Yaskawa INFORM job: DEMO_ROOF_UPPER_0625_3PAINT_27.JBI

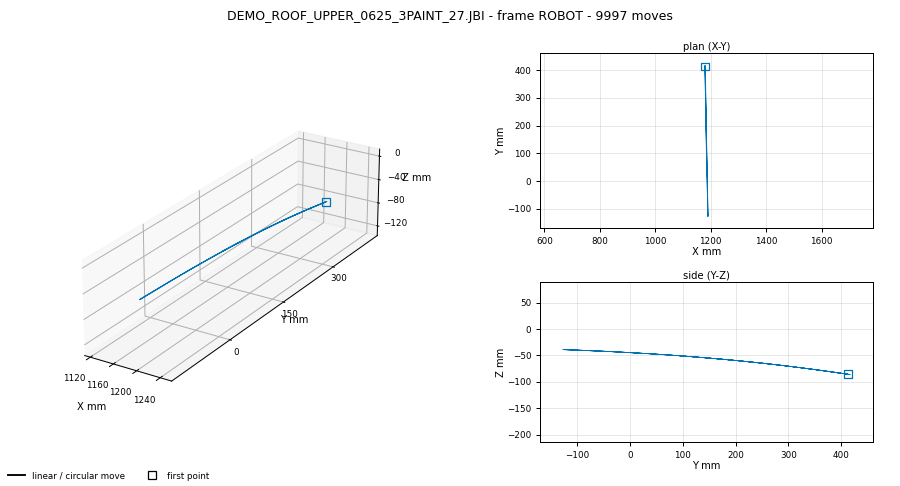
[picture p0: tool path of DEMO_ROOF_UPPER_0625_3PAINT_27.JBI in frame ROBOT, 9997 of 9997 moves have a stored position in this frame; points joined in program order, loops and branches not executed]
/JOB
//NAME DEMO_ROOF_UPPER_0625_3PAINT27
//POS
///NPOS 9997,0,0,0,0,0
///TOOL 0
///USER 0
///POSTYPE ROBOT
///RECTAN
///RCONF 1,0,0,0,0,0,0,0,0,0,0,0,0,0,0,0,0,0,0,0,0,0,0,0
C00000=1180.489,413.583,-85.570,-176.011,9.119,148.688
C00001=1180.493,413.335,-85.534,-176.011,9.117,148.687
C00002=1180.497,413.087,-85.498,-176.011,9.115,148.686
C00003=1180.501,412.840,-85.462,-176.011,9.113,148.686
C00004=1180.505,412.594,-85.426,-176.010,9.111,148.686
C00005=1180.509,412.346,-85.390,-176.010,9.109,148.685
C00006=1180.513,412.098,-85.354,-176.010,9.107,148.684
C00007=1180.517,411.851,-85.319,-176.010,9.105,148.684
C00008=1180.521,411.603,-85.282,-176.011,9.103,148.683
C00009=1180.525,411.356,-85.246,-176.010,9.101,148.683
C00010=1180.528,411.108,-85.211,-176.010,9.099,148.682
C00011=1180.532,410.861,-85.174,-176.010,9.097,148.682
C00012=1180.536,410.614,-85.138,-176.010,9.095,148.681
C00013=1180.540,410.367,-85.103,-176.009,9.093,148.680
C00014=1180.545,410.119,-85.067,-176.010,9.091,148.680
C00015=1180.548,409.872,-85.031,-176.009,9.089,148.679
C00016=1180.553,409.625,-84.995,-176.009,9.087,148.679
C00017=1180.556,409.377,-84.959,-176.009,9.085,148.678
C00018=1180.560,409.130,-84.924,-176.009,9.082,148.678
C00019=1180.564,408.882,-84.887,-176.009,9.081,148.677
C00020=1180.568,408.635,-84.851,-176.009,9.079,148.677
C00021=1180.572,408.388,-84.816,-176.009,9.076,148.676
C00022=1180.576,408.140,-84.780,-176.009,9.075,148.675
C00023=1180.580,407.893,-84.744,-176.009,9.072,148.675
C00024=1180.583,407.646,-84.708,-176.009,9.070,148.674
C00025=1180.588,407.398,-84.672,-176.009,9.068,148.674
C00026=1180.591,407.151,-84.636,-176.008,9.066,148.673
C00027=1180.595,406.903,-84.601,-176.009,9.064,148.672
C00028=1180.599,406.655,-84.565,-176.008,9.062,148.672
C00029=1180.603,406.409,-84.529,-176.008,9.060,148.671
C00030=1180.607,406.162,-84.493,-176.008,9.057,148.671
C00031=1180.611,405.914,-84.457,-176.008,9.056,148.670
C00032=1180.615,405.666,-84.422,-176.008,9.053,148.670
C00033=1180.619,405.419,-84.386,-176.008,9.051,148.669
C00034=1180.623,405.171,-84.350,-176.008,9.048,148.668
C00035=1180.627,404.924,-84.314,-176.008,9.047,148.668
C00036=1180.631,404.677,-84.278,-176.008,9.044,148.667
C00037=1180.635,404.429,-84.242,-176.008,9.042,148.667
C00038=1180.639,404.182,-84.207,-176.008,9.040,148.666
C00039=1180.643,403.934,-84.171,-176.008,9.037,148.665
C00040=1180.647,403.687,-84.135,-176.007,9.036,148.665
C00041=1180.650,403.440,-84.099,-176.008,9.033,148.664
C00042=1180.655,403.193,-84.064,-176.007,9.031,148.664
C00043=1180.659,402.945,-84.027,-176.008,9.029,148.663
C00044=1180.663,402.698,-83.992,-176.007,9.026,148.662
C00045=1180.666,402.450,-83.956,-176.008,9.024,148.662
C00046=1180.670,402.203,-83.921,-176.008,9.021,148.661
C00047=1180.674,401.955,-83.885,-176.007,9.020,148.661
C00048=1180.678,401.709,-83.849,-176.007,9.017,148.660
C00049=1180.682,401.461,-83.813,-176.007,9.015,148.659
C00050=1180.686,401.213,-83.777,-176.007,9.012,148.659
C00051=1180.690,400.966,-83.741,-176.007,9.010,148.658
C00052=1180.694,400.718,-83.706,-176.007,9.007,148.657
C00053=1180.697,400.471,-83.670,-176.008,9.005,148.657
C00054=1180.702,400.224,-83.635,-176.007,9.003,148.656
C00055=1180.706,399.976,-83.599,-176.008,9.000,148.656
C00056=1180.710,399.729,-83.564,-176.007,8.998,148.655
C00057=1180.714,399.481,-83.527,-176.008,8.996,148.654
C00058=1180.718,399.233,-83.492,-176.008,8.993,148.654
C00059=1180.721,398.987,-83.456,-176.007,8.990,148.653
C00060=1180.725,398.740,-83.420,-176.008,8.988,148.652
C00061=1180.730,398.492,-83.384,-176.007,8.986,148.652
C00062=1180.733,398.244,-83.349,-176.008,8.983,148.651
C00063=1180.737,397.997,-83.313,-176.008,8.981,148.650
C00064=1180.741,397.749,-83.278,-176.008,8.978,148.650
C00065=1180.746,397.502,-83.242,-176.008,8.976,148.649
C00066=1180.749,397.255,-83.206,-176.008,8.974,148.649
C00067=1180.753,397.007,-83.171,-176.008,8.970,148.648
C00068=1180.757,396.760,-83.135,-176.008,8.968,148.647
C00069=1180.761,396.512,-83.099,-176.008,8.965,148.647
C00070=1180.765,396.265,-83.064,-176.008,8.963,148.646
C00071=1180.769,396.018,-83.028,-176.008,8.961,148.645
C00072=1180.773,395.770,-82.993,-176.008,8.958,148.645
C00073=1180.776,395.523,-82.957,-176.009,8.955,148.644
C00074=1180.781,395.276,-82.921,-176.009,8.952,148.643
C00075=1180.785,395.028,-82.886,-176.009,8.950,148.643
C00076=1180.789,394.781,-82.850,-176.009,8.948,148.642
C00077=1180.792,394.533,-82.815,-176.009,8.945,148.641
C00078=1180.797,394.285,-82.779,-176.010,8.942,148.641
C00079=1180.801,394.038,-82.743,-176.009,8.939,148.640
C00080=1180.805,393.791,-82.708,-176.010,8.937,148.640
C00081=1180.808,393.543,-82.672,-176.010,8.934,148.639
C00082=1180.812,393.296,-82.637,-176.010,8.931,148.638
C00083=1180.816,393.048,-82.601,-176.010,8.929,148.638
C00084=1180.821,392.801,-82.565,-176.011,8.926,148.637
C00085=1180.824,392.554,-82.530,-176.011,8.923,148.636
C00086=1180.829,392.269,-82.490,-176.011,8.920,148.636
C00087=1180.833,391.986,-82.449,-176.012,8.916,148.635
C00088=1180.838,391.701,-82.408,-176.011,8.914,148.634
C00089=1180.842,391.417,-82.367,-176.012,8.911,148.633
C00090=1180.846,391.169,-82.332,-176.013,8.907,148.633
C00091=1180.850,390.922,-82.297,-176.013,8.905,148.632
C00092=1180.854,390.675,-82.261,-176.013,8.902,148.631
C00093=1180.859,390.427,-82.225,-176.014,8.899,148.631
C00094=1180.862,390.180,-82.190,-176.014,8.896,148.630
C00095=1180.866,389.933,-82.154,-176.014,8.894,148.630
C00096=1180.870,389.685,-82.119,-176.015,8.890,148.629
C00097=1180.874,389.438,-82.083,-176.015,8.888,148.628
C00098=1180.878,389.190,-82.049,-176.015,8.885,148.627
C00099=1180.882,388.943,-82.013,-176.016,8.882,148.627
C00100=1180.886,388.695,-81.978,-176.016,8.879,148.626
C00101=1180.890,388.448,-81.942,-176.017,8.876,148.626
C00102=1180.894,388.200,-81.906,-176.018,8.873,148.625
C00103=1180.898,387.953,-81.871,-176.017,8.870,148.624
C00104=1180.902,387.705,-81.836,-176.018,8.867,148.624
C00105=1180.906,387.458,-81.801,-176.019,8.864,148.623
C00106=1180.910,387.211,-81.765,-176.019,8.861,148.622
C00107=1180.914,386.963,-81.730,-176.020,8.858,148.622
C00108=1180.917,386.716,-81.694,-176.020,8.855,148.621
C00109=1180.921,386.468,-81.659,-176.021,8.852,148.620
C00110=1180.925,386.221,-81.624,-176.022,8.849,148.620
C00111=1180.929,385.973,-81.589,-176.022,8.845,148.619
C00112=1180.933,385.726,-81.553,-176.022,8.843,148.619
C00113=1180.938,385.478,-81.518,-176.023,8.840,148.618
C00114=1180.942,385.231,-81.483,-176.024,8.837,148.617
C00115=1180.945,384.983,-81.447,-176.024,8.834,148.617
C00116=1180.949,384.736,-81.411,-176.025,8.830,148.616
C00117=1180.954,384.488,-81.377,-176.026,8.827,148.615
C00118=1180.957,384.241,-81.341,-176.027,8.824,148.615
C00119=1180.961,383.993,-81.306,-176.028,8.821,148.614
C00120=1180.966,383.746,-81.271,-176.028,8.818,148.614
C00121=1180.969,383.498,-81.236,-176.029,8.815,148.613
C00122=1180.973,383.251,-81.200,-176.030,8.812,148.612
C00123=1180.977,383.003,-81.166,-176.031,8.809,148.612
C00124=1180.981,382.756,-81.130,-176.031,8.805,148.611
C00125=1180.985,382.508,-81.095,-176.032,8.802,148.611
C00126=1180.989,382.261,-81.060,-176.033,8.799,148.610
C00127=1180.993,382.014,-81.025,-176.034,8.795,148.609
C00128=1180.997,381.766,-80.989,-176.035,8.792,148.609
C00129=1181.001,381.519,-80.955,-176.036,8.789,148.608
C00130=1181.005,381.271,-80.919,-176.036,8.786,148.607
C00131=1181.009,381.024,-80.885,-176.037,8.783,148.607
C00132=1181.013,380.776,-80.849,-176.038,8.780,148.606
C00133=1181.017,380.529,-80.814,-176.039,8.776,148.606
C00134=1181.021,380.281,-80.779,-176.040,8.773,148.605
C00135=1181.025,380.034,-80.744,-176.041,8.769,148.604
C00136=1181.029,379.786,-80.709,-176.042,8.766,148.604
C00137=1181.033,379.539,-80.674,-176.044,8.763,148.603
C00138=1181.036,379.291,-80.639,-176.045,8.760,148.603
C00139=1181.040,379.044,-80.604,-176.045,8.757,148.602
C00140=1181.045,378.796,-80.569,-176.047,8.753,148.602
C00141=1181.048,378.549,-80.534,-176.048,8.750,148.601
C00142=1181.053,378.301,-80.499,-176.048,8.746,148.601
C00143=1181.057,378.054,-80.464,-176.050,8.743,148.600
C00144=1181.061,377.806,-80.429,-176.051,8.740,148.599
C00145=1181.065,377.559,-80.394,-176.052,8.736,148.599
C00146=1181.069,377.311,-80.359,-176.053,8.733,148.598
C00147=1181.073,377.064,-80.324,-176.054,8.730,148.598
C00148=1181.076,376.816,-80.290,-176.055,8.726,148.597
C00149=1181.081,376.569,-80.254,-176.057,8.723,148.597
C00150=1181.085,376.321,-80.220,-176.058,8.719,148.596
C00151=1181.088,376.073,-80.185,-176.059,8.716,148.595
C00152=1181.093,375.826,-80.150,-176.061,8.712,148.595
C00153=1181.097,375.578,-80.115,-176.062,8.709,148.594
C00154=1181.101,375.331,-80.080,-176.063,8.705,148.594
C00155=1181.104,375.083,-80.045,-176.064,8.702,148.593
C00156=1181.109,374.836,-80.011,-176.066,8.699,148.593
C00157=1181.112,374.589,-79.975,-176.066,8.695,148.592
C00158=1181.116,374.340,-79.940,-176.068,8.692,148.592
C00159=1181.121,374.093,-79.906,-176.070,8.688,148.591
C00160=1181.124,373.846,-79.871,-176.071,8.685,148.591
C00161=1181.128,373.598,-79.837,-176.072,8.681,148.590
C00162=1181.132,373.350,-79.802,-176.073,8.678,148.590
C00163=1181.137,373.103,-79.767,-176.075,8.674,148.589
C00164=1181.140,372.856,-79.732,-176.077,8.671,148.589
C00165=1181.145,372.608,-79.698,-176.077,8.668,148.588
C00166=1181.148,372.360,-79.663,-176.079,8.664,148.588
C00167=1181.153,372.113,-79.629,-176.081,8.661,148.587
C00168=1181.156,371.866,-79.594,-176.082,8.657,148.587
C00169=1181.161,371.618,-79.559,-176.084,8.654,148.586
C00170=1181.165,371.370,-79.524,-176.085,8.650,148.586
C00171=1181.169,371.123,-79.490,-176.087,8.646,148.585
C00172=1181.172,370.875,-79.455,-176.088,8.643,148.585
C00173=1181.177,370.628,-79.420,-176.090,8.640,148.584
C00174=1181.181,370.380,-79.386,-176.091,8.636,148.584
C00175=1181.184,370.133,-79.352,-176.093,8.633,148.583
C00176=1181.188,369.885,-79.317,-176.095,8.630,148.583
C00177=1181.193,369.637,-79.282,-176.096,8.626,148.582
C00178=1181.196,369.389,-79.248,-176.098,8.622,148.582
C00179=1181.200,369.143,-79.213,-176.100,8.618,148.581
C00180=1181.204,368.894,-79.178,-176.101,8.616,148.581
C00181=1181.208,368.647,-79.144,-176.103,8.612,148.581
C00182=1181.212,368.399,-79.109,-176.104,8.608,148.580
C00183=1181.217,368.152,-79.075,-176.106,8.604,148.580
C00184=1181.221,367.905,-79.041,-176.108,8.601,148.579
C00185=1181.225,367.657,-79.006,-176.109,8.598,148.579
C00186=1181.229,367.409,-78.972,-176.111,8.594,148.578
C00187=1181.232,367.161,-78.938,-176.113,8.591,148.578
C00188=1181.237,366.914,-78.903,-176.114,8.587,148.577
C00189=1181.240,366.666,-78.869,-176.116,8.584,148.577
C00190=1181.245,366.384,-78.829,-176.118,8.580,148.577
C00191=1181.249,366.103,-78.791,-176.120,8.575,148.576
C00192=1181.254,365.821,-78.752,-176.122,8.572,148.576
C00193=1181.258,365.540,-78.713,-176.125,8.567,148.575
C00194=1181.263,365.292,-78.678,-176.126,8.564,148.575
C00195=1181.267,365.045,-78.645,-176.128,8.561,148.574
C00196=1181.271,364.797,-78.610,-176.129,8.557,148.574
C00197=1181.275,364.550,-78.575,-176.131,8.554,148.573
C00198=1181.279,364.302,-78.541,-176.133,8.550,148.573
C00199=1181.283,364.054,-78.507,-176.135,8.547,148.573
C00200=1181.287,363.807,-78.473,-176.137,8.543,148.572
C00201=1181.291,363.558,-78.439,-176.139,8.540,148.572
C00202=1181.295,363.311,-78.405,-176.141,8.536,148.572
C00203=1181.298,363.064,-78.371,-176.143,8.532,148.571
C00204=1181.303,362.816,-78.336,-176.144,8.529,148.571
C00205=1181.307,362.569,-78.302,-176.147,8.525,148.570
C00206=1181.311,362.320,-78.268,-176.149,8.522,148.570
C00207=1181.315,362.073,-78.234,-176.150,8.518,148.570
C00208=1181.319,361.826,-78.200,-176.153,8.515,148.569
C00209=1181.323,361.578,-78.165,-176.154,8.511,148.569
C00210=1181.328,361.330,-78.132,-176.156,8.508,148.568
C00211=1181.331,361.083,-78.098,-176.159,8.504,148.568
C00212=1181.335,360.835,-78.064,-176.160,8.501,148.568
C00213=1181.339,360.588,-78.029,-176.162,8.497,148.567
C00214=1181.343,360.340,-77.996,-176.164,8.494,148.567
C00215=1181.347,360.092,-77.961,-176.166,8.490,148.567
C00216=1181.351,359.845,-77.927,-176.169,8.487,148.567
C00217=1181.355,359.597,-77.894,-176.170,8.483,148.566
C00218=1181.360,359.349,-77.860,-176.173,8.480,148.566
C00219=1181.363,359.101,-77.826,-176.174,8.476,148.565
C00220=1181.367,358.854,-77.792,-176.177,8.473,148.565
C00221=1181.372,358.606,-77.758,-176.178,8.469,148.565
C00222=1181.375,358.358,-77.724,-176.181,8.466,148.565
C00223=1181.379,358.111,-77.690,-176.183,8.462,148.564
C00224=1181.384,357.863,-77.657,-176.185,8.459,148.564
C00225=1181.388,357.616,-77.623,-176.187,8.456,148.564
C00226=1181.391,357.367,-77.589,-176.189,8.451,148.563
C00227=1181.396,357.120,-77.555,-176.192,8.448,148.563
C00228=1181.400,356.872,-77.522,-176.194,8.444,148.563
C00229=1181.404,356.625,-77.488,-176.196,8.441,148.562
C00230=1181.407,356.377,-77.454,-176.198,8.438,148.562
C00231=1181.412,356.129,-77.420,-176.200,8.434,148.562
C00232=1181.416,355.882,-77.387,-176.202,8.431,148.561
C00233=1181.420,355.634,-77.353,-176.204,8.428,148.561
C00234=1181.424,355.387,-77.320,-176.206,8.424,148.561
C00235=1181.428,355.139,-77.285,-176.208,8.421,148.561
C00236=1181.432,354.891,-77.252,-176.211,8.417,148.560
C00237=1181.436,354.643,-77.218,-176.213,8.414,148.560
C00238=1181.440,354.396,-77.185,-176.215,8.410,148.560
C00239=1181.444,354.148,-77.151,-176.217,8.407,148.559
C00240=1181.449,353.899,-77.117,-176.219,8.404,148.559
C00241=1181.452,353.652,-77.083,-176.221,8.400,148.559
C00242=1181.457,353.405,-77.050,-176.224,8.396,148.559
C00243=1181.461,353.157,-77.017,-176.226,8.393,148.558
C00244=1181.465,352.910,-76.983,-176.229,8.389,148.558
C00245=1181.469,352.662,-76.950,-176.230,8.386,148.558
C00246=1181.473,352.413,-76.916,-176.233,8.382,148.557
C00247=1181.477,352.166,-76.883,-176.235,8.379,148.557
C00248=1181.481,351.919,-76.849,-176.237,8.376,148.557
C00249=1181.485,351.671,-76.816,-176.239,8.372,148.557
C00250=1181.489,351.423,-76.783,-176.241,8.369,148.556
C00251=1181.493,351.175,-76.750,-176.243,8.366,148.556
C00252=1181.497,350.928,-76.716,-176.246,8.362,148.556
C00253=1181.501,350.680,-76.682,-176.248,8.359,148.556
C00254=1181.505,350.432,-76.649,-176.250,8.356,148.556
C00255=1181.510,350.184,-76.615,-176.253,8.352,148.555
C00256=1181.514,349.936,-76.582,-176.254,8.349,148.555
C00257=1181.518,349.689,-76.549,-176.257,8.345,148.555
C00258=1181.522,349.441,-76.516,-176.259,8.342,148.554
C00259=1181.526,349.193,-76.483,-176.261,8.339,148.554
C00260=1181.530,348.946,-76.449,-176.263,8.335,148.554
C00261=1181.534,348.698,-76.416,-176.266,8.332,148.554
C00262=1181.538,348.451,-76.382,-176.268,8.329,148.554
C00263=1181.543,348.203,-76.349,-176.270,8.325,148.553
C00264=1181.547,347.955,-76.316,-176.273,8.321,148.553
C00265=1181.550,347.707,-76.283,-176.275,8.318,148.553
C00266=1181.554,347.459,-76.249,-176.278,8.315,148.553
C00267=1181.559,347.211,-76.216,-176.279,8.311,148.552
C00268=1181.563,346.963,-76.183,-176.282,8.308,148.552
C00269=1181.567,346.716,-76.150,-176.284,8.304,148.552
C00270=1181.571,346.468,-76.117,-176.286,8.301,148.552
C00271=1181.575,346.220,-76.084,-176.288,8.298,148.551
C00272=1181.579,345.973,-76.050,-176.291,8.294,148.551
C00273=1181.584,345.724,-76.018,-176.293,8.291,148.551
C00274=1181.587,345.477,-75.985,-176.295,8.288,148.551
C00275=1181.591,345.229,-75.952,-176.297,8.285,148.550
C00276=1181.595,344.981,-75.919,-176.300,8.281,148.550
C00277=1181.599,344.734,-75.886,-176.302,8.278,148.550
C00278=1181.604,344.486,-75.853,-176.304,8.275,148.550
C00279=1181.608,344.238,-75.820,-176.307,8.272,148.550
C00280=1181.612,343.990,-75.787,-176.309,8.268,148.550
C00281=1181.616,343.742,-75.754,-176.311,8.265,148.549
C00282=1181.620,343.494,-75.721,-176.314,8.262,148.549
C00283=1181.624,343.247,-75.688,-176.316,8.258,148.549
C00284=1181.628,342.999,-75.655,-176.318,8.255,148.549
C00285=1181.632,342.751,-75.623,-176.320,8.252,148.549
C00286=1181.637,342.503,-75.590,-176.323,8.248,148.548
C00287=1181.641,342.256,-75.557,-176.325,8.245,148.548
C00288=1181.645,342.008,-75.524,-176.327,8.242,148.548
C00289=1181.649,341.760,-75.492,-176.330,8.238,148.548
C00290=1181.653,341.513,-75.459,-176.332,8.235,148.547
C00291=1181.657,341.265,-75.426,-176.335,8.232,148.547
C00292=1181.662,341.016,-75.393,-176.337,8.229,148.547
C00293=1181.666,340.769,-75.360,-176.339,8.226,148.547
C00294=1181.670,340.490,-75.323,-176.342,8.221,148.547
C00295=1181.674,340.211,-75.286,-176.344,8.218,148.547
C00296=1181.680,339.931,-75.250,-176.347,8.214,148.546
C00297=1181.684,339.653,-75.213,-176.350,8.211,148.546
C00298=1181.688,339.405,-75.180,-176.352,8.208,148.546
C00299=1181.693,339.157,-75.148,-176.354,8.204,148.546
C00300=1181.696,338.909,-75.115,-176.356,8.201,148.546
C00301=1181.700,338.662,-75.082,-176.359,8.198,148.545
C00302=1181.705,338.413,-75.050,-176.361,8.194,148.545
C00303=1181.709,338.167,-75.017,-176.364,8.191,148.545
C00304=1181.713,337.918,-74.985,-176.366,8.188,148.545
C00305=1181.717,337.671,-74.952,-176.368,8.185,148.545
C00306=1181.721,337.422,-74.920,-176.370,8.181,148.545
C00307=1181.726,337.174,-74.888,-176.373,8.178,148.545
C00308=1181.730,336.926,-74.854,-176.375,8.175,148.544
C00309=1181.733,336.678,-74.823,-176.378,8.172,148.544
C00310=1181.738,336.431,-74.790,-176.380,8.168,148.544
C00311=1181.742,336.183,-74.758,-176.383,8.165,148.544
C00312=1181.746,335.936,-74.725,-176.385,8.162,148.544
C00313=1181.750,335.687,-74.692,-176.387,8.159,148.543
C00314=1181.754,335.439,-74.661,-176.389,8.156,148.543
C00315=1181.758,335.191,-74.627,-176.392,8.153,148.543
C00316=1181.763,334.944,-74.596,-176.394,8.149,148.543
C00317=1181.767,334.696,-74.563,-176.397,8.146,148.543
C00318=1181.770,334.448,-74.531,-176.399,8.143,148.543
C00319=1181.775,334.200,-74.498,-176.402,8.140,148.543
C00320=1181.779,333.953,-74.467,-176.404,8.136,148.542
C00321=1181.783,333.705,-74.434,-176.406,8.133,148.542
C00322=1181.788,333.457,-74.401,-176.409,8.130,148.542
C00323=1181.792,333.209,-74.370,-176.411,8.127,148.542
C00324=1181.796,332.960,-74.337,-176.413,8.123,148.542
C00325=1181.800,332.713,-74.305,-176.416,8.120,148.542
C00326=1181.804,332.465,-74.273,-176.418,8.117,148.542
C00327=1181.808,332.217,-74.241,-176.421,8.114,148.541
C00328=1181.812,331.969,-74.209,-176.423,8.111,148.541
C00329=1181.817,331.721,-74.177,-176.426,8.107,148.541
C00330=1181.820,331.474,-74.144,-176.428,8.104,148.541
C00331=1181.825,331.226,-74.112,-176.431,8.101,148.541
C00332=1181.828,330.978,-74.080,-176.433,8.098,148.541
C00333=1181.833,330.730,-74.048,-176.435,8.094,148.541
C00334=1181.837,330.482,-74.016,-176.438,8.091,148.541
C00335=1181.841,330.234,-73.984,-176.440,8.088,148.540
C00336=1181.846,329.986,-73.952,-176.443,8.085,148.540
C00337=1181.850,329.738,-73.920,-176.445,8.083,148.540
C00338=1181.854,329.490,-73.888,-176.447,8.079,148.540
C00339=1181.858,329.242,-73.856,-176.449,8.076,148.540
C00340=1181.862,328.994,-73.824,-176.452,8.073,148.540
C00341=1181.867,328.746,-73.792,-176.454,8.070,148.540
C00342=1181.870,328.498,-73.760,-176.457,8.067,148.540
C00343=1181.875,328.251,-73.729,-176.459,8.063,148.539
C00344=1181.879,328.002,-73.696,-176.462,8.060,148.539
C00345=1181.883,327.754,-73.664,-176.464,8.057,148.539
C00346=1181.887,327.507,-73.633,-176.467,8.054,148.539
C00347=1181.891,327.259,-73.600,-176.469,8.051,148.539
C00348=1181.896,327.011,-73.569,-176.472,8.048,148.539
C00349=1181.899,326.763,-73.537,-176.474,8.044,148.539
C00350=1181.904,326.515,-73.505,-176.476,8.041,148.539
C00351=1181.908,326.268,-73.473,-176.479,8.038,148.539
C00352=1181.912,326.020,-73.441,-176.481,8.035,148.538
C00353=1181.916,325.772,-73.409,-176.484,8.032,148.538
C00354=1181.921,325.523,-73.378,-176.486,8.028,148.538
C00355=1181.925,325.275,-73.346,-176.489,8.025,148.538
C00356=1181.929,325.028,-73.315,-176.491,8.022,148.538
C00357=1181.933,324.780,-73.283,-176.494,8.019,148.538
C00358=1181.937,324.531,-73.250,-176.496,8.016,148.538
C00359=1181.942,324.284,-73.220,-176.499,8.013,148.538
C00360=1181.945,324.035,-73.188,-176.500,8.010,148.538
C00361=1181.950,323.788,-73.156,-176.503,8.007,148.538
C00362=1181.953,323.540,-73.125,-176.505,8.004,148.537
C00363=1181.957,323.291,-73.093,-176.508,8.001,148.537
C00364=1181.963,323.044,-73.061,-176.510,7.998,148.537
C00365=1181.966,322.796,-73.030,-176.513,7.995,148.537
C00366=1181.971,322.548,-72.998,-176.515,7.991,148.537
C00367=1181.975,322.300,-72.967,-176.518,7.988,148.537
C00368=1181.979,322.052,-72.935,-176.520,7.985,148.537
C00369=1181.983,321.804,-72.904,-176.523,7.982,148.537
C00370=1181.987,321.556,-72.872,-176.525,7.979,148.537
C00371=1181.991,321.308,-72.841,-176.528,7.976,148.537
C00372=1181.996,321.059,-72.809,-176.531,7.973,148.537
C00373=1182.000,320.812,-72.778,-176.533,7.970,148.536
C00374=1182.004,320.564,-72.746,-176.536,7.967,148.536
C00375=1182.008,320.316,-72.715,-176.538,7.963,148.536
C00376=1182.012,320.068,-72.683,-176.540,7.961,148.536
C00377=1182.017,319.820,-72.653,-176.542,7.958,148.536
C00378=1182.020,319.572,-72.621,-176.545,7.955,148.536
C00379=1182.025,319.324,-72.590,-176.547,7.951,148.536
C00380=1182.029,319.076,-72.558,-176.550,7.948,148.536
C00381=1182.033,318.828,-72.527,-176.553,7.945,148.536
C00382=1182.037,318.580,-72.495,-176.555,7.942,148.536
C00383=1182.042,318.332,-72.465,-176.558,7.939,148.536
C00384=1182.045,318.084,-72.433,-176.560,7.936,148.535
C00385=1182.050,317.836,-72.402,-176.563,7.933,148.535
C00386=1182.054,317.588,-72.370,-176.566,7.930,148.535
C00387=1182.058,317.340,-72.339,-176.568,7.926,148.535
C00388=1182.063,317.092,-72.309,-176.570,7.923,148.535
C00389=1182.067,316.844,-72.277,-176.572,7.921,148.535
C00390=1182.071,316.596,-72.246,-176.575,7.918,148.535
C00391=1182.075,316.348,-72.214,-176.578,7.915,148.535
C00392=1182.079,316.100,-72.184,-176.580,7.912,148.535
C00393=1182.083,315.851,-72.152,-176.583,7.909,148.535
C00394=1182.088,315.604,-72.121,-176.585,7.905,148.535
C00395=1182.092,315.357,-72.091,-176.588,7.902,148.535
C00396=1182.096,315.108,-72.060,-176.590,7.899,148.535
C00397=1182.100,314.860,-72.029,-176.593,7.896,148.535
C00398=1182.105,314.583,-71.994,-176.595,7.893,148.535
C00399=1182.109,314.307,-71.959,-176.598,7.890,148.535
C00400=1182.114,314.030,-71.924,-176.601,7.886,148.534
C00401=1182.119,313.753,-71.890,-176.604,7.883,148.534
C00402=1182.123,313.505,-71.859,-176.606,7.880,148.534
C00403=1182.128,313.257,-71.828,-176.609,7.877,148.534
C00404=1182.132,313.010,-71.797,-176.611,7.874,148.534
C00405=1182.136,312.761,-71.766,-176.614,7.871,148.534
C00406=1182.140,312.513,-71.735,-176.617,7.868,148.534
C00407=1182.144,312.264,-71.704,-176.619,7.864,148.534
C00408=1182.149,312.016,-71.674,-176.621,7.862,148.534
C00409=1182.152,311.769,-71.643,-176.624,7.859,148.534
C00410=1182.156,311.521,-71.612,-176.626,7.856,148.534
C00411=1182.161,311.273,-71.581,-176.629,7.853,148.534
C00412=1182.166,311.025,-71.550,-176.631,7.850,148.534
C00413=1182.169,310.777,-71.520,-176.634,7.847,148.534
C00414=1182.174,310.529,-71.489,-176.636,7.844,148.534
C00415=1182.178,310.281,-71.458,-176.639,7.841,148.534
C00416=1182.183,310.033,-71.427,-176.641,7.837,148.534
C00417=1182.186,309.784,-71.397,-176.644,7.835,148.534
C00418=1182.191,309.536,-71.366,-176.646,7.832,148.534
C00419=1182.195,309.288,-71.335,-176.649,7.829,148.533
C00420=1182.199,309.040,-71.304,-176.651,7.826,148.533
C00421=1182.203,308.792,-71.274,-176.654,7.823,148.533
C00422=1182.208,308.544,-71.243,-176.657,7.820,148.534
C00423=1182.212,308.296,-71.212,-176.659,7.816,148.533
C00424=1182.216,308.048,-71.182,-176.662,7.813,148.533
C00425=1182.220,307.800,-71.151,-176.664,7.810,148.533
C00426=1182.225,307.552,-71.120,-176.667,7.808,148.533
C00427=1182.229,307.304,-71.091,-176.669,7.805,148.533
C00428=1182.233,307.055,-71.060,-176.672,7.802,148.533
C00429=1182.237,306.807,-71.030,-176.674,7.799,148.533
C00430=1182.242,306.559,-70.999,-176.677,7.796,148.533
C00431=1182.246,306.311,-70.968,-176.679,7.793,148.533
C00432=1182.249,306.063,-70.937,-176.682,7.790,148.533
C00433=1182.254,305.814,-70.907,-176.685,7.787,148.533
C00434=1182.258,305.567,-70.877,-176.687,7.785,148.533
C00435=1182.263,305.319,-70.846,-176.689,7.781,148.533
C00436=1182.267,305.071,-70.816,-176.692,7.778,148.533
C00437=1182.271,304.823,-70.785,-176.695,7.775,148.533
C00438=1182.276,304.574,-70.755,-176.697,7.772,148.533
C00439=1182.280,304.326,-70.725,-176.700,7.769,148.533
C00440=1182.284,304.078,-70.694,-176.702,7.766,148.533
C00441=1182.288,303.830,-70.665,-176.704,7.764,148.533
C00442=1182.293,303.582,-70.634,-176.707,7.761,148.533
C00443=1182.296,303.334,-70.603,-176.709,7.757,148.533
C00444=1182.301,303.085,-70.573,-176.712,7.754,148.533
C00445=1182.305,302.838,-70.543,-176.715,7.751,148.533
C00446=1182.310,302.590,-70.512,-176.718,7.748,148.533
C00447=1182.314,302.341,-70.483,-176.720,7.745,148.533
C00448=1182.318,302.093,-70.452,-176.722,7.743,148.533
C00449=1182.322,301.846,-70.422,-176.725,7.740,148.533
C00450=1182.327,301.596,-70.392,-176.727,7.737,148.533
C00451=1182.330,301.349,-70.361,-176.730,7.734,148.533
C00452=1182.335,301.100,-70.331,-176.733,7.731,148.533
C00453=1182.339,300.853,-70.301,-176.735,7.728,148.533
C00454=1182.343,300.604,-70.272,-176.737,7.726,148.533
C00455=1182.348,300.356,-70.241,-176.740,7.723,148.533
C00456=1182.352,300.108,-70.212,-176.743,7.720,148.533
C00457=1182.357,299.860,-70.181,-176.745,7.717,148.533
C00458=1182.361,299.612,-70.151,-176.748,7.713,148.533
C00459=1182.365,299.364,-70.121,-176.750,7.710,148.533
C00460=1182.369,299.115,-70.091,-176.753,7.707,148.533
C00461=1182.373,298.867,-70.061,-176.755,7.705,148.533
C00462=1182.377,298.619,-70.031,-176.758,7.702,148.533
C00463=1182.382,298.370,-70.001,-176.761,7.699,148.533
C00464=1182.386,298.123,-69.971,-176.763,7.696,148.533
C00465=1182.390,297.875,-69.942,-176.766,7.693,148.533
C00466=1182.395,297.627,-69.911,-176.768,7.690,148.533
C00467=1182.399,297.378,-69.881,-176.771,7.688,148.533
C00468=1182.403,297.130,-69.852,-176.773,7.685,148.533
C00469=1182.408,296.882,-69.821,-176.776,7.682,148.533
C00470=1182.412,296.634,-69.792,-176.779,7.679,148.533
C00471=1182.416,296.386,-69.762,-176.781,7.675,148.533
C00472=1182.420,296.138,-69.732,-176.783,7.673,148.533
C00473=1182.425,295.889,-69.702,-176.786,7.670,148.533
C00474=1182.429,295.641,-69.672,-176.789,7.667,148.533
C00475=1182.433,295.393,-69.643,-176.791,7.664,148.533
C00476=1182.437,295.145,-69.613,-176.794,7.661,148.533
C00477=1182.442,294.897,-69.583,-176.797,7.658,148.533
C00478=1182.446,294.648,-69.553,-176.798,7.656,148.533
C00479=1182.451,294.400,-69.524,-176.801,7.653,148.533
C00480=1182.454,294.152,-69.494,-176.804,7.650,148.533
C00481=1182.459,293.904,-69.464,-176.807,7.647,148.533
C00482=1182.463,293.656,-69.434,-176.809,7.644,148.533
C00483=1182.468,293.407,-69.405,-176.812,7.642,148.533
C00484=1182.472,293.159,-69.375,-176.814,7.639,148.533
C00485=1182.476,292.911,-69.346,-176.817,7.636,148.533
C00486=1182.480,292.662,-69.316,-176.820,7.633,148.533
C00487=1182.484,292.415,-69.286,-176.822,7.629,148.533
C00488=1182.488,292.167,-69.257,-176.824,7.627,148.533
C00489=1182.493,291.918,-69.227,-176.827,7.624,148.533
C00490=1182.497,291.670,-69.197,-176.830,7.621,148.533
C00491=1182.502,291.421,-69.168,-176.832,7.618,148.533
C00492=1182.506,291.173,-69.138,-176.835,7.615,148.533
C00493=1182.510,290.925,-69.109,-176.837,7.613,148.533
C00494=1182.515,290.677,-69.080,-176.840,7.610,148.533
C00495=1182.519,290.429,-69.050,-176.843,7.607,148.533
C00496=1182.523,290.181,-69.021,-176.845,7.604,148.533
C00497=1182.527,289.933,-68.992,-176.848,7.601,148.533
C00498=1182.531,289.684,-68.962,-176.850,7.599,148.533
C00499=1182.536,289.436,-68.933,-176.852,7.596,148.533
C00500=1182.540,289.188,-68.903,-176.855,7.593,148.533
C00501=1182.544,288.939,-68.874,-176.858,7.590,148.533
C00502=1182.550,288.665,-68.841,-176.861,7.587,148.533
C00503=1182.553,288.390,-68.809,-176.863,7.584,148.533
C00504=1182.559,288.116,-68.776,-176.866,7.581,148.533
C00505=1182.563,287.841,-68.744,-176.869,7.578,148.533
C00506=1182.567,287.592,-68.715,-176.872,7.575,148.533
C00507=1182.572,287.345,-68.686,-176.874,7.572,148.533
C00508=1182.576,287.097,-68.656,-176.877,7.569,148.533
C00509=1182.580,286.848,-68.627,-176.880,7.566,148.533
C00510=1182.585,286.599,-68.598,-176.882,7.563,148.533
C00511=1182.589,286.351,-68.569,-176.885,7.561,148.533
C00512=1182.593,286.103,-68.539,-176.887,7.558,148.533
C00513=1182.598,285.855,-68.510,-176.890,7.555,148.533
C00514=1182.602,285.607,-68.481,-176.892,7.552,148.533
C00515=1182.607,285.358,-68.452,-176.895,7.549,148.534
C00516=1182.611,285.110,-68.423,-176.898,7.546,148.534
C00517=1182.615,284.862,-68.393,-176.900,7.543,148.534
C00518=1182.620,284.614,-68.365,-176.903,7.541,148.534
C00519=1182.624,284.365,-68.336,-176.905,7.538,148.534
C00520=1182.628,284.117,-68.307,-176.908,7.535,148.534
C00521=1182.632,283.868,-68.278,-176.911,7.532,148.534
C00522=1182.637,283.621,-68.249,-176.913,7.530,148.534
C00523=1182.641,283.372,-68.219,-176.916,7.527,148.534
C00524=1182.646,283.124,-68.191,-176.918,7.524,148.534
C00525=1182.649,282.876,-68.162,-176.921,7.521,148.534
C00526=1182.654,282.627,-68.133,-176.923,7.519,148.534
C00527=1182.659,282.379,-68.104,-176.926,7.516,148.534
C00528=1182.663,282.131,-68.074,-176.929,7.513,148.534
C00529=1182.667,281.882,-68.046,-176.931,7.510,148.534
C00530=1182.671,281.635,-68.017,-176.934,7.508,148.534
C00531=1182.676,281.386,-67.988,-176.936,7.505,148.534
C00532=1182.680,281.138,-67.959,-176.939,7.502,148.534
C00533=1182.685,280.889,-67.931,-176.942,7.499,148.534
C00534=1182.688,280.641,-67.902,-176.944,7.497,148.534
C00535=1182.693,280.393,-67.873,-176.947,7.494,148.534
C00536=1182.697,280.144,-67.844,-176.949,7.491,148.534
C00537=1182.702,279.896,-67.815,-176.952,7.488,148.534
C00538=1182.706,279.648,-67.786,-176.954,7.486,148.535
C00539=1182.710,279.399,-67.758,-176.957,7.483,148.535
C00540=1182.715,279.151,-67.729,-176.960,7.480,148.535
C00541=1182.719,278.903,-67.700,-176.962,7.477,148.535
C00542=1182.723,278.654,-67.672,-176.965,7.474,148.535
C00543=1182.728,278.407,-67.643,-176.967,7.471,148.535
C00544=1182.732,278.158,-67.614,-176.970,7.468,148.535
C00545=1182.736,277.909,-67.586,-176.972,7.466,148.535
C00546=1182.741,277.662,-67.557,-176.975,7.463,148.535
C00547=1182.745,277.413,-67.528,-176.978,7.460,148.535
C00548=1182.749,277.164,-67.500,-176.980,7.457,148.535
C00549=1182.754,276.917,-67.471,-176.983,7.455,148.535
C00550=1182.758,276.668,-67.442,-176.985,7.452,148.535
C00551=1182.763,276.420,-67.414,-176.988,7.450,148.535
C00552=1182.767,276.171,-67.386,-176.991,7.447,148.535
C00553=1182.771,275.923,-67.356,-176.993,7.444,148.536
C00554=1182.775,275.675,-67.329,-176.996,7.441,148.536
C00555=1182.780,275.426,-67.300,-176.998,7.439,148.536
C00556=1182.784,275.177,-67.271,-177.001,7.436,148.536
C00557=1182.788,274.930,-67.243,-177.004,7.433,148.536
C00558=1182.793,274.681,-67.214,-177.006,7.430,148.536
C00559=1182.797,274.433,-67.186,-177.009,7.428,148.536
C00560=1182.801,274.184,-67.157,-177.011,7.425,148.536
C00561=1182.806,273.937,-67.130,-177.014,7.422,148.536
C00562=1182.810,273.688,-67.101,-177.016,7.420,148.536
C00563=1182.814,273.440,-67.072,-177.019,7.417,148.536
C00564=1182.819,273.192,-67.044,-177.022,7.414,148.536
C00565=1182.823,272.943,-67.016,-177.024,7.412,148.536
C00566=1182.828,272.695,-66.987,-177.027,7.409,148.536
C00567=1182.831,272.446,-66.959,-177.030,7.406,148.536
C00568=1182.836,272.198,-66.931,-177.032,7.404,148.537
C00569=1182.840,271.949,-66.903,-177.035,7.401,148.537
C00570=1182.845,271.701,-66.874,-177.037,7.398,148.537
C00571=1182.849,271.453,-66.846,-177.040,7.395,148.537
C00572=1182.853,271.205,-66.818,-177.042,7.393,148.537
C00573=1182.858,270.956,-66.790,-177.045,7.390,148.537
C00574=1182.862,270.708,-66.762,-177.048,7.387,148.537
C00575=1182.867,270.459,-66.733,-177.050,7.385,148.537
C00576=1182.871,270.211,-66.705,-177.053,7.382,148.537
C00577=1182.875,269.963,-66.677,-177.056,7.379,148.537
C00578=1182.880,269.714,-66.649,-177.058,7.377,148.537
C00579=1182.884,269.466,-66.621,-177.061,7.374,148.537
C00580=1182.889,269.218,-66.592,-177.063,7.371,148.537
C00581=1182.893,268.969,-66.564,-177.066,7.369,148.538
C00582=1182.897,268.721,-66.536,-177.068,7.366,148.538
C00583=1182.902,268.472,-66.508,-177.072,7.363,148.538
C00584=1182.906,268.224,-66.480,-177.074,7.361,148.538
C00585=1182.910,267.975,-66.452,-177.076,7.358,148.538
C00586=1182.915,267.727,-66.424,-177.079,7.356,148.538
C00587=1182.919,267.479,-66.396,-177.081,7.353,148.538
C00588=1182.923,267.231,-66.368,-177.084,7.350,148.538
C00589=1182.928,266.982,-66.340,-177.086,7.348,148.538
C00590=1182.932,266.733,-66.312,-177.089,7.345,148.538
C00591=1182.936,266.485,-66.284,-177.092,7.342,148.539
C00592=1182.940,266.237,-66.256,-177.094,7.340,148.539
C00593=1182.946,265.988,-66.229,-177.097,7.337,148.539
C00594=1182.950,265.740,-66.201,-177.100,7.334,148.539
C00595=1182.954,265.492,-66.173,-177.102,7.332,148.539
C00596=1182.958,265.244,-66.145,-177.105,7.329,148.539
C00597=1182.963,264.994,-66.117,-177.108,7.326,148.539
C00598=1182.967,264.746,-66.089,-177.110,7.324,148.539
C00599=1182.972,264.498,-66.061,-177.113,7.321,148.539
C00600=1182.976,264.249,-66.034,-177.115,7.319,148.539
C00601=1182.980,264.001,-66.006,-177.118,7.316,148.539
C00602=1182.985,263.753,-65.978,-177.121,7.313,148.540
C00603=1182.989,263.504,-65.950,-177.123,7.311,148.540
C00604=1182.993,263.256,-65.923,-177.126,7.308,148.540
C00605=1182.998,263.007,-65.895,-177.128,7.305,148.540
C00606=1183.003,262.734,-65.865,-177.131,7.302,148.540
C00607=1183.007,262.461,-65.834,-177.134,7.300,148.540
C00608=1183.013,262.188,-65.804,-177.137,7.297,148.540
C00609=1183.017,261.915,-65.774,-177.139,7.294,148.540
C00610=1183.022,261.667,-65.745,-177.143,7.292,148.541
C00611=1183.026,261.419,-65.718,-177.145,7.289,148.541
C00612=1183.030,261.170,-65.690,-177.147,7.287,148.541
C00613=1183.035,260.922,-65.663,-177.150,7.284,148.541
C00614=1183.039,260.674,-65.635,-177.153,7.281,148.541
C00615=1183.043,260.424,-65.608,-177.156,7.279,148.541
C00616=1183.048,260.177,-65.580,-177.158,7.276,148.541
C00617=1183.052,259.928,-65.553,-177.160,7.274,148.541
C00618=1183.057,259.680,-65.525,-177.163,7.271,148.541
C00619=1183.061,259.431,-65.498,-177.166,7.268,148.542
C00620=1183.065,259.183,-65.471,-177.169,7.266,148.542
C00621=1183.070,258.935,-65.443,-177.171,7.263,148.542
C00622=1183.074,258.686,-65.416,-177.173,7.261,148.542
C00623=1183.078,258.438,-65.388,-177.176,7.258,148.542
C00624=1183.083,258.189,-65.361,-177.179,7.255,148.542
C00625=1183.087,257.941,-65.334,-177.182,7.253,148.542
C00626=1183.092,257.693,-65.306,-177.184,7.250,148.542
C00627=1183.096,257.444,-65.279,-177.186,7.248,148.542
C00628=1183.100,257.195,-65.251,-177.190,7.245,148.543
C00629=1183.105,256.947,-65.224,-177.192,7.243,148.543
C00630=1183.109,256.699,-65.197,-177.195,7.240,148.543
C00631=1183.113,256.449,-65.169,-177.197,7.237,148.543
C00632=1183.118,256.201,-65.142,-177.200,7.235,148.543
C00633=1183.122,255.953,-65.114,-177.203,7.232,148.543
C00634=1183.127,255.705,-65.087,-177.205,7.230,148.543
C00635=1183.132,255.456,-65.060,-177.208,7.227,148.543
C00636=1183.136,255.207,-65.033,-177.210,7.225,148.544
C00637=1183.140,254.958,-65.006,-177.213,7.222,148.544
C00638=1183.145,254.711,-64.978,-177.216,7.219,148.544
C00639=1183.149,254.462,-64.952,-177.218,7.218,148.544
C00640=1183.153,254.214,-64.924,-177.221,7.215,148.544
C00641=1183.157,253.965,-64.897,-177.223,7.212,148.544
C00642=1183.162,253.716,-64.870,-177.226,7.209,148.544
C00643=1183.167,253.468,-64.843,-177.229,7.208,148.545
C00644=1183.171,253.219,-64.816,-177.231,7.205,148.545
C00645=1183.175,252.971,-64.789,-177.233,7.202,148.545
C00646=1183.180,252.723,-64.762,-177.237,7.200,148.545
C00647=1183.184,252.475,-64.735,-177.239,7.197,148.545
C00648=1183.188,252.225,-64.707,-177.242,7.195,148.545
C00649=1183.193,251.977,-64.680,-177.244,7.192,148.545
C00650=1183.197,251.729,-64.654,-177.247,7.190,148.546
C00651=1183.202,251.480,-64.627,-177.250,7.187,148.546
C00652=1183.206,251.232,-64.599,-177.252,7.185,148.546
C00653=1183.211,250.983,-64.572,-177.255,7.182,148.546
C00654=1183.216,250.735,-64.545,-177.257,7.180,148.546
C00655=1183.220,250.487,-64.519,-177.260,7.177,148.546
C00656=1183.224,250.238,-64.492,-177.263,7.175,148.546
C00657=1183.228,249.989,-64.464,-177.265,7.172,148.547
C00658=1183.233,249.740,-64.437,-177.267,7.170,148.547
C00659=1183.237,249.492,-64.412,-177.271,7.167,148.547
C00660=1183.242,249.243,-64.385,-177.273,7.164,148.547
C00661=1183.246,248.995,-64.357,-177.276,7.162,148.547
C00662=1183.250,248.746,-64.331,-177.279,7.160,148.547
C00663=1183.255,248.498,-64.304,-177.281,7.157,148.547
C00664=1183.260,248.249,-64.277,-177.284,7.154,148.547
C00665=1183.264,248.001,-64.250,-177.286,7.153,148.548
C00666=1183.268,247.753,-64.223,-177.289,7.150,148.548
C00667=1183.273,247.504,-64.197,-177.291,7.148,148.548
C00668=1183.277,247.255,-64.171,-177.294,7.145,148.548
C00669=1183.282,247.007,-64.143,-177.297,7.143,148.548
C00670=1183.286,246.758,-64.116,-177.299,7.140,148.548
C00671=1183.291,246.510,-64.091,-177.302,7.138,148.549
C00672=1183.295,246.261,-64.064,-177.305,7.135,148.549
C00673=1183.299,246.013,-64.037,-177.307,7.133,148.549
C00674=1183.304,245.764,-64.010,-177.310,7.130,148.549
C00675=1183.309,245.515,-63.984,-177.312,7.128,148.549
C00676=1183.313,245.267,-63.957,-177.316,7.125,148.550
C00677=1183.317,245.019,-63.930,-177.318,7.123,148.550
C00678=1183.321,244.770,-63.904,-177.320,7.120,148.550
C00679=1183.326,244.521,-63.877,-177.323,7.118,148.550
C00680=1183.330,244.273,-63.851,-177.326,7.115,148.550
C00681=1183.335,244.025,-63.824,-177.328,7.113,148.550
C00682=1183.340,243.776,-63.798,-177.331,7.111,148.550
C00683=1183.344,243.527,-63.771,-177.333,7.108,148.551
C00684=1183.349,243.278,-63.745,-177.337,7.106,148.551
C00685=1183.353,243.030,-63.718,-177.339,7.104,148.551
C00686=1183.357,242.782,-63.691,-177.341,7.101,148.551
C00687=1183.362,242.533,-63.665,-177.344,7.099,148.551
C00688=1183.366,242.284,-63.638,-177.347,7.096,148.551
C00689=1183.370,242.035,-63.613,-177.349,7.094,148.552
C00690=1183.374,241.787,-63.586,-177.352,7.092,148.552
C00691=1183.379,241.538,-63.560,-177.354,7.089,148.552
C00692=1183.383,241.290,-63.533,-177.357,7.087,148.552
C00693=1183.388,241.041,-63.507,-177.360,7.084,148.552
C00694=1183.393,240.793,-63.481,-177.362,7.082,148.553
C00695=1183.398,240.544,-63.455,-177.365,7.079,148.553
C00696=1183.402,240.296,-63.428,-177.367,7.077,148.553
C00697=1183.407,240.047,-63.402,-177.371,7.075,148.553
C00698=1183.410,239.799,-63.375,-177.373,7.072,148.553
C00699=1183.415,239.550,-63.350,-177.376,7.070,148.553
C00700=1183.419,239.302,-63.322,-177.378,7.068,148.554
C00701=1183.424,239.053,-63.297,-177.381,7.065,148.554
C00702=1183.428,238.804,-63.271,-177.384,7.063,148.554
C00703=1183.433,238.556,-63.244,-177.386,7.061,148.554
C00704=1183.437,238.307,-63.218,-177.389,7.058,148.554
C00705=1183.442,238.058,-63.192,-177.391,7.056,148.554
C00706=1183.446,237.810,-63.166,-177.394,7.053,148.555
C00707=1183.450,237.561,-63.140,-177.396,7.051,148.555
C00708=1183.455,237.312,-63.114,-177.400,7.048,148.555
C00709=1183.460,237.065,-63.087,-177.402,7.046,148.555
C00710=1183.465,236.793,-63.059,-177.405,7.044,148.555
C00711=1183.469,236.521,-63.031,-177.408,7.041,148.556
C00712=1183.474,236.249,-63.002,-177.410,7.039,148.556
C00713=1183.479,235.978,-62.973,-177.414,7.036,148.556
C00714=1183.484,235.730,-62.948,-177.416,7.033,148.556
C00715=1183.489,235.481,-62.922,-177.419,7.031,148.557
C00716=1183.493,235.232,-62.896,-177.421,7.029,148.557
C00717=1183.497,234.984,-62.869,-177.424,7.027,148.557
C00718=1183.501,234.735,-62.844,-177.427,7.025,148.557
C00719=1183.506,234.487,-62.818,-177.429,7.022,148.557
C00720=1183.511,234.238,-62.792,-177.432,7.020,148.557
C00721=1183.515,233.989,-62.766,-177.434,7.018,148.558
C00722=1183.519,233.740,-62.740,-177.437,7.015,148.558
C00723=1183.524,233.493,-62.714,-177.440,7.013,148.558
C00724=1183.529,233.243,-62.688,-177.443,7.010,148.558
C00725=1183.533,232.995,-62.662,-177.445,7.008,148.558
C00726=1183.537,232.746,-62.636,-177.448,7.005,148.559
C00727=1183.542,232.498,-62.611,-177.450,7.003,148.559
C00728=1183.546,232.249,-62.585,-177.453,7.001,148.559
C00729=1183.550,232.000,-62.560,-177.456,6.998,148.559
C00730=1183.555,231.751,-62.533,-177.458,6.997,148.559
C00731=1183.560,231.503,-62.508,-177.461,6.994,148.560
C00732=1183.564,231.254,-62.482,-177.464,6.992,148.560
C00733=1183.569,231.005,-62.456,-177.466,6.990,148.560
C00734=1183.573,230.757,-62.431,-177.469,6.987,148.560
C00735=1183.578,230.508,-62.405,-177.472,6.985,148.561
C00736=1183.582,230.260,-62.379,-177.474,6.983,148.561
C00737=1183.586,230.011,-62.354,-177.477,6.980,148.561
C00738=1183.591,229.763,-62.328,-177.479,6.978,148.561
C00739=1183.595,229.514,-62.303,-177.483,6.976,148.561
C00740=1183.600,229.265,-62.276,-177.485,6.974,148.561
C00741=1183.605,229.017,-62.251,-177.487,6.972,148.562
C00742=1183.609,228.768,-62.225,-177.490,6.969,148.562
C00743=1183.613,228.519,-62.199,-177.493,6.967,148.562
C00744=1183.618,228.271,-62.174,-177.496,6.964,148.562
C00745=1183.623,228.022,-62.149,-177.498,6.962,148.563
C00746=1183.627,227.773,-62.123,-177.500,6.960,148.563
C00747=1183.632,227.525,-62.098,-177.504,6.957,148.563
C00748=1183.636,227.276,-62.072,-177.506,6.956,148.563
C00749=1183.640,227.027,-62.046,-177.508,6.953,148.563
C00750=1183.645,226.779,-62.021,-177.512,6.951,148.564
C00751=1183.650,226.529,-61.996,-177.514,6.949,148.564
C00752=1183.654,226.281,-61.970,-177.517,6.946,148.564
C00753=1183.659,226.033,-61.945,-177.519,6.944,148.564
C00754=1183.663,225.784,-61.919,-177.522,6.942,148.565
C00755=1183.668,225.535,-61.894,-177.525,6.939,148.565
C00756=1183.672,225.286,-61.869,-177.527,6.937,148.565
C00757=1183.676,225.038,-61.843,-177.530,6.935,148.565
C00758=1183.681,224.790,-61.818,-177.533,6.932,148.565
C00759=1183.685,224.540,-61.793,-177.535,6.931,148.566
C00760=1183.690,224.292,-61.768,-177.537,6.929,148.566
C00761=1183.694,224.043,-61.742,-177.541,6.926,148.566
C00762=1183.699,223.795,-61.717,-177.543,6.924,148.566
C00763=1183.703,223.546,-61.691,-177.546,6.922,148.567
C00764=1183.708,223.297,-61.666,-177.549,6.919,148.567
C00765=1183.713,223.048,-61.641,-177.551,6.917,148.567
C00766=1183.717,222.799,-61.615,-177.554,6.915,148.567
C00767=1183.721,222.552,-61.590,-177.557,6.913,148.568
C00768=1183.726,222.302,-61.565,-177.559,6.911,148.568
C00769=1183.731,222.054,-61.540,-177.562,6.909,148.568
C00770=1183.735,221.805,-61.515,-177.564,6.906,148.568
C00771=1183.740,221.557,-61.490,-177.567,6.904,148.569
C00772=1183.744,221.307,-61.465,-177.570,6.902,148.569
C00773=1183.748,221.059,-61.440,-177.572,6.899,148.569
C00774=1183.753,220.810,-61.415,-177.575,6.897,148.569
C00775=1183.758,220.562,-61.389,-177.578,6.896,148.570
C00776=1183.762,220.313,-61.364,-177.580,6.893,148.570
C00777=1183.766,220.065,-61.340,-177.583,6.891,148.570
C00778=1183.771,219.815,-61.314,-177.585,6.889,148.570
C00779=1183.776,219.567,-61.289,-177.589,6.886,148.570
C00780=1183.780,219.318,-61.264,-177.591,6.884,148.571
C00781=1183.784,219.070,-61.239,-177.593,6.882,148.571
C00782=1183.789,218.820,-61.214,-177.597,6.879,148.571
C00783=1183.794,218.572,-61.189,-177.599,6.878,148.572
C00784=1183.798,218.323,-61.164,-177.601,6.876,148.572
C00785=1183.803,218.075,-61.140,-177.605,6.873,148.572
C00786=1183.807,217.826,-61.114,-177.607,6.871,148.572
C00787=1183.812,217.577,-61.089,-177.609,6.869,148.572
C00788=1183.816,217.329,-61.064,-177.613,6.866,148.573
C00789=1183.821,217.080,-61.039,-177.615,6.864,148.573
C00790=1183.825,216.830,-61.014,-177.618,6.862,148.573
C00791=1183.829,216.583,-60.990,-177.620,6.861,148.573
C00792=1183.834,216.334,-60.965,-177.623,6.858,148.574
C00793=1183.839,216.084,-60.940,-177.626,6.856,148.574
C00794=1183.843,215.837,-60.915,-177.628,6.854,148.574
C00795=1183.848,215.587,-60.890,-177.631,6.851,148.574
C00796=1183.853,215.338,-60.865,-177.634,6.849,148.575
C00797=1183.857,215.090,-60.841,-177.636,6.847,148.575
C00798=1183.861,214.841,-60.816,-177.639,6.844,148.575
C00799=1183.866,214.593,-60.792,-177.642,6.843,148.575
C00800=1183.870,214.343,-60.767,-177.644,6.841,148.576
C00801=1183.875,214.095,-60.742,-177.647,6.839,148.576
C00802=1183.880,213.846,-60.718,-177.650,6.836,148.576
C00803=1183.884,213.597,-60.692,-177.652,6.834,148.576
C00804=1183.888,213.349,-60.668,-177.655,6.832,148.577
C00805=1183.894,213.100,-60.643,-177.657,6.830,148.577
C00806=1183.897,212.851,-60.619,-177.660,6.828,148.577
C00807=1183.902,212.603,-60.594,-177.663,6.826,148.578
C00808=1183.906,212.353,-60.570,-177.665,6.824,148.578
C00809=1183.911,212.105,-60.545,-177.669,6.821,148.578
C00810=1183.916,211.857,-60.520,-177.671,6.819,148.578
C00811=1183.920,211.607,-60.495,-177.673,6.817,148.578
C00812=1183.925,211.359,-60.471,-177.676,6.815,148.579
C00813=1183.930,211.110,-60.446,-177.679,6.813,148.579
C00814=1183.934,210.839,-60.419,-177.682,6.811,148.579
C00815=1183.940,210.569,-60.393,-177.685,6.808,148.580
C00816=1183.945,210.298,-60.367,-177.687,6.806,148.580
C00817=1183.950,210.028,-60.340,-177.691,6.804,148.580
C00818=1183.954,209.779,-60.316,-177.693,6.802,148.581
C00819=1183.958,209.531,-60.291,-177.696,6.800,148.581
C00820=1183.963,209.282,-60.267,-177.699,6.797,148.581
C00821=1183.967,209.033,-60.242,-177.701,6.795,148.581
C00822=1183.972,208.784,-60.218,-177.704,6.793,148.582
C00823=1183.976,208.536,-60.194,-177.706,6.791,148.582
C00824=1183.982,208.287,-60.169,-177.709,6.789,148.582
C00825=1183.985,208.038,-60.145,-177.712,6.787,148.582
C00826=1183.990,207.790,-60.120,-177.715,6.785,148.583
C00827=1183.995,207.541,-60.096,-177.717,6.783,148.583
C00828=1184.000,207.292,-60.072,-177.720,6.780,148.583
C00829=1184.004,207.042,-60.047,-177.723,6.778,148.584
C00830=1184.009,206.794,-60.023,-177.725,6.777,148.584
C00831=1184.013,206.546,-59.999,-177.728,6.775,148.584
C00832=1184.018,206.297,-59.975,-177.731,6.772,148.584
C00833=1184.022,206.048,-59.950,-177.733,6.770,148.585
C00834=1184.027,205.799,-59.927,-177.736,6.768,148.585
C00835=1184.032,205.550,-59.902,-177.738,6.766,148.585
C00836=1184.036,205.302,-59.878,-177.741,6.764,148.585
C00837=1184.041,205.053,-59.854,-177.744,6.762,148.586
C00838=1184.045,204.804,-59.829,-177.746,6.760,148.586
C00839=1184.050,204.555,-59.806,-177.749,6.758,148.586
C00840=1184.054,204.306,-59.781,-177.752,6.756,148.587
C00841=1184.059,204.058,-59.757,-177.755,6.753,148.587
C00842=1184.064,203.809,-59.733,-177.757,6.751,148.587
C00843=1184.068,203.560,-59.709,-177.760,6.749,148.587
C00844=1184.072,203.311,-59.685,-177.762,6.748,148.588
C00845=1184.077,203.063,-59.661,-177.765,6.746,148.588
C00846=1184.082,202.813,-59.637,-177.768,6.743,148.588
C00847=1184.086,202.565,-59.613,-177.771,6.741,148.589
C00848=1184.091,202.316,-59.589,-177.773,6.739,148.589
C00849=1184.095,202.067,-59.565,-177.776,6.737,148.589
C00850=1184.099,201.818,-59.541,-177.779,6.736,148.590
C00851=1184.104,201.570,-59.516,-177.781,6.733,148.590
C00852=1184.109,201.321,-59.493,-177.784,6.731,148.590
C00853=1184.113,201.072,-59.469,-177.787,6.729,148.590
C00854=1184.118,200.823,-59.445,-177.789,6.727,148.591
C00855=1184.123,200.575,-59.421,-177.791,6.725,148.591
C00856=1184.127,200.326,-59.397,-177.795,6.723,148.591
C00857=1184.132,200.076,-59.373,-177.797,6.721,148.591
C00858=1184.136,199.828,-59.349,-177.800,6.719,148.592
C00859=1184.141,199.579,-59.326,-177.803,6.717,148.592
C00860=1184.145,199.330,-59.302,-177.805,6.715,148.592
C00861=1184.150,199.081,-59.278,-177.808,6.713,148.593
C00862=1184.154,198.833,-59.254,-177.811,6.711,148.593
C00863=1184.159,198.584,-59.231,-177.813,6.709,148.593
C00864=1184.163,198.335,-59.207,-177.816,6.707,148.593
C00865=1184.168,198.086,-59.183,-177.818,6.705,148.594
C00866=1184.173,197.838,-59.159,-177.821,6.703,148.594
C00867=1184.178,197.589,-59.135,-177.824,6.701,148.594
C00868=1184.183,197.340,-59.112,-177.827,6.699,148.595
C00869=1184.187,197.091,-59.088,-177.829,6.697,148.595
C00870=1184.191,196.841,-59.064,-177.832,6.695,148.595
C00871=1184.196,196.593,-59.040,-177.834,6.693,148.596
C00872=1184.200,196.344,-59.017,-177.837,6.691,148.596
C00873=1184.205,196.095,-58.993,-177.840,6.689,148.596
C00874=1184.209,195.847,-58.969,-177.843,6.687,148.597
C00875=1184.214,195.598,-58.946,-177.845,6.685,148.597
C00876=1184.219,195.349,-58.923,-177.848,6.683,148.597
C00877=1184.223,195.100,-58.898,-177.850,6.681,148.597
C00878=1184.228,194.851,-58.875,-177.853,6.679,148.598
C00879=1184.233,194.602,-58.852,-177.856,6.677,148.598
C00880=1184.237,194.354,-58.828,-177.859,6.675,148.598
C00881=1184.242,194.105,-58.804,-177.861,6.673,148.599
C00882=1184.246,193.856,-58.781,-177.864,6.671,148.599
C00883=1184.251,193.607,-58.758,-177.867,6.669,148.599
C00884=1184.255,193.358,-58.734,-177.869,6.667,148.600
C00885=1184.260,193.109,-58.710,-177.872,6.666,148.600
C00886=1184.265,192.860,-58.687,-177.874,6.663,148.600
C00887=1184.269,192.611,-58.664,-177.877,6.661,148.600
C00888=1184.274,192.362,-58.641,-177.880,6.659,148.601
C00889=1184.279,192.115,-58.617,-177.883,6.657,148.601
C00890=1184.283,191.866,-58.594,-177.885,6.655,148.602
C00891=1184.288,191.617,-58.570,-177.888,6.654,148.602
C00892=1184.293,191.368,-58.547,-177.890,6.652,148.602
C00893=1184.297,191.118,-58.524,-177.893,6.650,148.602
C00894=1184.302,190.869,-58.500,-177.896,6.647,148.603
C00895=1184.307,190.620,-58.477,-177.899,6.645,148.603
C00896=1184.310,190.372,-58.453,-177.901,6.644,148.603
C00897=1184.315,190.123,-58.430,-177.904,6.642,148.604
C00898=1184.320,189.874,-58.407,-177.907,6.640,148.604
C00899=1184.325,189.625,-58.383,-177.909,6.638,148.604
C00900=1184.329,189.376,-58.360,-177.912,6.636,148.605
C00901=1184.334,189.127,-58.337,-177.914,6.634,148.605
C00902=1184.338,188.879,-58.314,-177.917,6.632,148.605
C00903=1184.343,188.630,-58.291,-177.920,6.630,148.606
C00904=1184.348,188.381,-58.267,-177.923,6.628,148.606
C00905=1184.353,188.132,-58.244,-177.925,6.626,148.606
C00906=1184.357,187.883,-58.221,-177.928,6.624,148.606
C00907=1184.361,187.634,-58.198,-177.930,6.622,148.607
C00908=1184.366,187.385,-58.175,-177.933,6.621,148.607
C00909=1184.371,187.136,-58.151,-177.936,6.619,148.608
C00910=1184.376,186.888,-58.128,-177.938,6.617,148.608
C00911=1184.380,186.639,-58.105,-177.941,6.615,148.608
C00912=1184.385,186.390,-58.082,-177.944,6.613,148.609
C00913=1184.389,186.141,-58.059,-177.947,6.611,148.609
C00914=1184.394,185.892,-58.037,-177.950,6.609,148.609
C00915=1184.398,185.643,-58.013,-177.952,6.607,148.609
C00916=1184.404,185.394,-57.990,-177.954,6.605,148.610
C00917=1184.408,185.145,-57.967,-177.957,6.603,148.610
C00918=1184.413,184.876,-57.943,-177.960,6.601,148.610
C00919=1184.418,184.606,-57.918,-177.963,6.599,148.611
C00920=1184.423,184.337,-57.893,-177.966,6.597,148.611
C00921=1184.428,184.067,-57.868,-177.968,6.595,148.611
C00922=1184.433,183.818,-57.845,-177.971,6.594,148.612
C00923=1184.437,183.569,-57.822,-177.974,6.592,148.612
C00924=1184.441,183.320,-57.799,-177.976,6.590,148.613
C00925=1184.446,183.071,-57.775,-177.980,6.587,148.613
C00926=1184.451,182.822,-57.754,-177.982,6.586,148.613
C00927=1184.456,182.573,-57.730,-177.985,6.584,148.614
C00928=1184.460,182.325,-57.707,-177.988,6.582,148.614
C00929=1184.464,182.076,-57.684,-177.990,6.580,148.614
C00930=1184.470,181.827,-57.662,-177.993,6.578,148.615
C00931=1184.474,181.578,-57.639,-177.996,6.577,148.615
C00932=1184.479,181.329,-57.616,-177.998,6.574,148.615
C00933=1184.483,181.080,-57.594,-178.001,6.573,148.616
C00934=1184.488,180.831,-57.571,-178.003,6.571,148.616
C00935=1184.492,180.583,-57.548,-178.006,6.569,148.616
C00936=1184.497,180.333,-57.525,-178.009,6.567,148.617
C00937=1184.502,180.084,-57.502,-178.011,6.566,148.617
C00938=1184.506,179.836,-57.479,-178.014,6.564,148.617
C00939=1184.511,179.586,-57.457,-178.017,6.562,148.618
C00940=1184.515,179.338,-57.434,-178.019,6.560,148.618
C00941=1184.521,179.089,-57.412,-178.022,6.558,148.618
C00942=1184.525,178.840,-57.389,-178.025,6.556,148.619
C00943=1184.530,178.591,-57.366,-178.028,6.554,148.619
C00944=1184.534,178.341,-57.344,-178.030,6.552,148.619
C00945=1184.539,178.093,-57.321,-178.033,6.550,148.620
C00946=1184.543,177.844,-57.299,-178.035,6.548,148.620
C00947=1184.547,177.595,-57.276,-178.038,6.547,148.620
C00948=1184.553,177.346,-57.253,-178.041,6.545,148.621
C00949=1184.557,177.097,-57.231,-178.043,6.543,148.621
C00950=1184.562,176.848,-57.208,-178.046,6.541,148.621
C00951=1184.567,176.600,-57.186,-178.049,6.539,148.622
C00952=1184.572,176.350,-57.163,-178.051,6.538,148.622
C00953=1184.576,176.101,-57.140,-178.054,6.536,148.622
C00954=1184.580,175.853,-57.119,-178.057,6.534,148.623
C00955=1184.585,175.604,-57.095,-178.059,6.532,148.623
C00956=1184.589,175.354,-57.073,-178.062,6.531,148.624
C00957=1184.595,175.105,-57.051,-178.065,6.529,148.624
C00958=1184.599,174.857,-57.028,-178.067,6.527,148.624
C00959=1184.604,174.608,-57.006,-178.070,6.525,148.625
C00960=1184.609,174.359,-56.983,-178.073,6.523,148.625
C00961=1184.613,174.110,-56.961,-178.075,6.522,148.625
C00962=1184.618,173.861,-56.939,-178.078,6.520,148.626
C00963=1184.622,173.612,-56.916,-178.081,6.518,148.626
C00964=1184.627,173.363,-56.894,-178.083,6.516,148.626
C00965=1184.632,173.114,-56.872,-178.086,6.514,148.627
C00966=1184.636,172.865,-56.849,-178.089,6.513,148.627
C00967=1184.641,172.616,-56.827,-178.092,6.511,148.628
C00968=1184.645,172.367,-56.805,-178.094,6.509,148.628
C00969=1184.651,172.119,-56.782,-178.097,6.507,148.628
C00970=1184.655,171.869,-56.760,-178.100,6.506,148.629
C00971=1184.659,171.620,-56.738,-178.102,6.504,148.629
C00972=1184.665,171.371,-56.716,-178.105,6.502,148.629
C00973=1184.669,171.122,-56.693,-178.108,6.500,148.630
C00974=1184.674,170.874,-56.671,-178.110,6.498,148.630
C00975=1184.678,170.624,-56.649,-178.113,6.497,148.630
C00976=1184.683,170.375,-56.627,-178.116,6.495,148.631
C00977=1184.688,170.126,-56.605,-178.118,6.493,148.631
C00978=1184.692,169.878,-56.583,-178.121,6.491,148.632
C00979=1184.697,169.629,-56.561,-178.124,6.490,148.632
C00980=1184.702,169.380,-56.538,-178.126,6.488,148.632
C00981=1184.706,169.130,-56.516,-178.129,6.486,148.633
C00982=1184.711,168.882,-56.495,-178.132,6.484,148.633
C00983=1184.716,168.632,-56.472,-178.134,6.482,148.633
C00984=1184.720,168.384,-56.451,-178.137,6.481,148.634
C00985=1184.725,168.135,-56.427,-178.140,6.479,148.634
C00986=1184.730,167.886,-56.406,-178.142,6.477,148.635
C00987=1184.734,167.637,-56.384,-178.145,6.475,148.635
C00988=1184.739,167.388,-56.362,-178.148,6.474,148.635
C00989=1184.743,167.139,-56.340,-178.150,6.472,148.636
C00990=1184.748,166.890,-56.318,-178.153,6.471,148.636
C00991=1184.753,166.640,-56.296,-178.155,6.469,148.636
C00992=1184.758,166.392,-56.274,-178.158,6.467,148.637
C00993=1184.762,166.142,-56.252,-178.161,6.466,148.637
C00994=1184.767,165.894,-56.230,-178.163,6.464,148.637
C00995=1184.772,165.644,-56.208,-178.166,6.462,148.638
C00996=1184.776,165.396,-56.187,-178.169,6.460,148.638
C00997=1184.781,165.147,-56.164,-178.171,6.458,148.639
C00998=1184.786,164.898,-56.143,-178.174,6.457,148.639
C00999=1184.790,164.649,-56.121,-178.177,6.455,148.639
C01000=1184.795,164.400,-56.099,-178.179,6.453,148.640
C01001=1184.800,164.151,-56.077,-178.182,6.451,148.640
C01002=1184.804,163.902,-56.055,-178.185,6.450,148.640
C01003=1184.809,163.653,-56.033,-178.187,6.448,148.641
C01004=1184.814,163.403,-56.012,-178.190,6.446,148.641
C01005=1184.819,163.154,-55.990,-178.193,6.444,148.642
C01006=1184.824,162.906,-55.968,-178.195,6.442,148.642
C01007=1184.828,162.656,-55.946,-178.198,6.441,148.642
C01008=1184.833,162.408,-55.925,-178.200,6.440,148.643
C01009=1184.837,162.158,-55.903,-178.203,6.438,148.643
C01010=1184.842,161.910,-55.881,-178.206,6.436,148.643
C01011=1184.847,161.661,-55.860,-178.209,6.435,148.644
C01012=1184.852,161.411,-55.838,-178.211,6.433,148.644
C01013=1184.856,161.163,-55.816,-178.214,6.431,148.645
C01014=1184.861,160.913,-55.794,-178.217,6.429,148.645
C01015=1184.865,160.665,-55.773,-178.219,6.428,148.646
C01016=1184.870,160.416,-55.752,-178.222,6.426,148.646
C01017=1184.874,160.166,-55.730,-178.225,6.424,148.646
C01018=1184.879,159.918,-55.708,-178.227,6.422,148.647
C01019=1184.884,159.669,-55.687,-178.230,6.421,148.647
C01020=1184.889,159.419,-55.665,-178.232,6.420,148.647
C01021=1184.893,159.170,-55.644,-178.235,6.418,148.648
C01022=1184.899,158.901,-55.620,-178.238,6.415,148.648
C01023=1184.903,158.633,-55.597,-178.241,6.414,148.649
C01024=1184.909,158.363,-55.573,-178.244,6.412,148.649
C01025=1184.914,158.094,-55.551,-178.247,6.410,148.649
C01026=1184.918,157.846,-55.529,-178.249,6.409,148.650
C01027=1184.924,157.596,-55.508,-178.252,6.407,148.650
C01028=1184.928,157.347,-55.486,-178.255,6.405,148.651
C01029=1184.933,157.098,-55.464,-178.257,6.404,148.651
C01030=1184.937,156.849,-55.444,-178.260,6.403,148.652
C01031=1184.942,156.601,-55.422,-178.263,6.401,148.652
C01032=1184.946,156.351,-55.400,-178.265,6.399,148.652
C01033=1184.951,156.102,-55.379,-178.268,6.397,148.653
C01034=1184.956,155.853,-55.358,-178.271,6.396,148.653
C01035=1184.961,155.603,-55.336,-178.274,6.394,148.653
C01036=1184.965,155.355,-55.315,-178.276,6.392,148.654
C01037=1184.970,155.106,-55.294,-178.279,6.390,148.654
C01038=1184.975,154.857,-55.273,-178.281,6.389,148.655
C01039=1184.980,154.607,-55.251,-178.284,6.387,148.655
C01040=1184.985,154.359,-55.229,-178.287,6.386,148.656
C01041=1184.989,154.110,-55.209,-178.290,6.384,148.656
C01042=1184.994,153.861,-55.187,-178.292,6.383,148.656
C01043=1184.998,153.611,-55.166,-178.295,6.381,148.657
C01044=1185.003,153.362,-55.144,-178.298,6.379,148.657
C01045=1185.008,153.114,-55.124,-178.300,6.377,148.657
C01046=1185.013,152.865,-55.102,-178.302,6.376,148.658
C01047=1185.018,152.616,-55.081,-178.305,6.375,148.658
C01048=1185.021,152.367,-55.060,-178.308,6.373,148.659
C01049=1185.026,152.117,-55.039,-178.311,6.371,148.659
C01050=1185.032,151.868,-55.018,-178.314,6.370,148.660
C01051=1185.037,151.619,-54.996,-178.316,6.368,148.660
C01052=1185.041,151.370,-54.976,-178.319,6.366,148.660
C01053=1185.046,151.121,-54.955,-178.321,6.365,148.661
C01054=1185.050,150.872,-54.933,-178.324,6.363,148.661
C01055=1185.055,150.623,-54.913,-178.326,6.362,148.661
C01056=1185.060,150.374,-54.892,-178.329,6.360,148.662
C01057=1185.065,150.125,-54.870,-178.332,6.358,148.662
C01058=1185.069,149.876,-54.850,-178.335,6.357,148.663
C01059=1185.074,149.626,-54.828,-178.337,6.356,148.663
C01060=1185.079,149.377,-54.807,-178.340,6.354,148.664
C01061=1185.083,149.129,-54.786,-178.342,6.352,148.664
C01062=1185.088,148.879,-54.765,-178.345,6.350,148.664
C01063=1185.093,148.631,-54.744,-178.348,6.349,148.665
C01064=1185.098,148.382,-54.723,-178.351,6.347,148.665
C01065=1185.103,148.132,-54.702,-178.353,6.346,148.666
C01066=1185.107,147.883,-54.681,-178.356,6.344,148.666
C01067=1185.112,147.634,-54.660,-178.359,6.343,148.667
C01068=1185.116,147.385,-54.639,-178.361,6.341,148.667
C01069=1185.121,147.136,-54.618,-178.364,6.339,148.667
C01070=1185.126,146.887,-54.598,-178.367,6.337,148.668
C01071=1185.131,146.638,-54.577,-178.369,6.337,148.668
C01072=1185.136,146.388,-54.556,-178.372,6.335,148.669
C01073=1185.140,146.140,-54.535,-178.375,6.333,148.669
C01074=1185.145,145.891,-54.514,-178.377,6.332,148.669
C01075=1185.150,145.642,-54.494,-178.380,6.330,148.670
C01076=1185.154,145.392,-54.472,-178.383,6.328,148.670
C01077=1185.159,145.143,-54.452,-178.385,6.327,148.671
C01078=1185.164,144.894,-54.431,-178.388,6.326,148.671
C01079=1185.168,144.645,-54.411,-178.391,6.324,148.672
C01080=1185.174,144.396,-54.390,-178.393,6.322,148.672
C01081=1185.178,144.147,-54.369,-178.396,6.320,148.672
C01082=1185.183,143.897,-54.348,-178.398,6.319,148.673
C01083=1185.188,143.648,-54.328,-178.401,6.318,148.673
C01084=1185.192,143.400,-54.307,-178.404,6.316,148.674
C01085=1185.197,143.151,-54.286,-178.407,6.314,148.674
C01086=1185.201,142.902,-54.266,-178.409,6.313,148.674
C01087=1185.206,142.653,-54.245,-178.411,6.312,148.675
C01088=1185.211,142.404,-54.224,-178.414,6.310,148.675
C01089=1185.216,142.154,-54.203,-178.417,6.309,148.676
C01090=1185.221,141.905,-54.183,-178.420,6.307,148.676
C01091=1185.225,141.656,-54.162,-178.422,6.306,148.677
C01092=1185.230,141.407,-54.142,-178.425,6.304,148.677
C01093=1185.235,141.158,-54.122,-178.428,6.302,148.677
C01094=1185.240,140.908,-54.101,-178.431,6.301,148.678
C01095=1185.244,140.659,-54.081,-178.433,6.299,148.678
C01096=1185.249,140.411,-54.060,-178.435,6.298,148.679
C01097=1185.254,140.161,-54.039,-178.438,6.297,148.679
C01098=1185.259,139.912,-54.019,-178.441,6.295,148.680
C01099=1185.263,139.663,-53.998,-178.444,6.293,148.680
C01100=1185.268,139.414,-53.977,-178.446,6.292,148.681
C01101=1185.273,139.165,-53.957,-178.449,6.291,148.681
C01102=1185.277,138.916,-53.937,-178.452,6.289,148.681
C01103=1185.283,138.666,-53.916,-178.454,6.287,148.682
C01104=1185.287,138.417,-53.896,-178.457,6.286,148.682
C01105=1185.291,138.168,-53.876,-178.460,6.285,148.683
C01106=1185.297,137.919,-53.855,-178.462,6.283,148.683
C01107=1185.301,137.670,-53.834,-178.465,6.281,148.684
C01108=1185.306,137.421,-53.815,-178.468,6.280,148.684
C01109=1185.310,137.172,-53.794,-178.470,6.279,148.685
C01110=1185.315,136.922,-53.773,-178.473,6.277,148.685
C01111=1185.320,136.673,-53.753,-178.476,6.275,148.685
C01112=1185.325,136.425,-53.734,-178.478,6.274,148.686
C01113=1185.330,136.175,-53.713,-178.480,6.273,148.686
C01114=1185.335,135.926,-53.692,-178.484,6.271,148.687
C01115=1185.339,135.677,-53.672,-178.486,6.270,148.687
C01116=1185.344,135.428,-53.652,-178.489,6.268,148.688
C01117=1185.348,135.179,-53.632,-178.491,6.267,148.688
C01118=1185.354,134.930,-53.611,-178.494,6.265,148.689
C01119=1185.358,134.680,-53.591,-178.497,6.264,148.689
C01120=1185.363,134.431,-53.571,-178.500,6.262,148.689
C01121=1185.367,134.182,-53.551,-178.502,6.261,148.690
C01122=1185.372,133.933,-53.531,-178.505,6.260,148.690
C01123=1185.378,133.684,-53.510,-178.508,6.258,148.691
C01124=1185.382,133.435,-53.491,-178.510,6.256,148.691
C01125=1185.387,133.186,-53.470,-178.512,6.255,148.692
C01126=1185.393,132.917,-53.449,-178.516,6.254,148.692
C01127=1185.397,132.649,-53.427,-178.518,6.252,148.693
C01128=1185.403,132.380,-53.405,-178.521,6.250,148.693
C01129=1185.407,132.112,-53.383,-178.524,6.249,148.694
C01130=1185.412,131.862,-53.364,-178.527,6.247,148.694
C01131=1185.417,131.613,-53.343,-178.529,6.246,148.694
C01132=1185.421,131.363,-53.324,-178.532,6.245,148.695
C01133=1185.427,131.115,-53.303,-178.535,6.243,148.695
C01134=1185.432,130.865,-53.283,-178.538,6.241,148.696
C01135=1185.436,130.616,-53.263,-178.540,6.240,148.696
C01136=1185.441,130.367,-53.243,-178.543,6.239,148.697
C01137=1185.445,130.118,-53.223,-178.546,6.237,148.697
C01138=1185.451,129.869,-53.204,-178.548,6.236,148.698
C01139=1185.455,129.620,-53.183,-178.550,6.234,148.698
C01140=1185.460,129.371,-53.164,-178.554,6.233,148.699
C01141=1185.464,129.122,-53.143,-178.556,6.231,148.699
C01142=1185.469,128.872,-53.124,-178.558,6.230,148.699
C01143=1185.474,128.623,-53.104,-178.562,6.229,148.700
C01144=1185.479,128.374,-53.084,-178.564,6.227,148.700
C01145=1185.484,128.125,-53.064,-178.566,6.226,148.701
C01146=1185.488,127.876,-53.044,-178.569,6.225,148.701
C01147=1185.493,127.627,-53.025,-178.572,6.223,148.702
C01148=1185.498,127.377,-53.005,-178.574,6.222,148.702
C01149=1185.503,127.128,-52.985,-178.577,6.220,148.703
C01150=1185.507,126.879,-52.965,-178.580,6.219,148.703
C01151=1185.513,126.630,-52.946,-178.583,6.217,148.704
C01152=1185.517,126.381,-52.925,-178.585,6.216,148.704
C01153=1185.522,126.131,-52.906,-178.588,6.215,148.704
C01154=1185.527,125.882,-52.886,-178.591,6.213,148.705
C01155=1185.532,125.634,-52.866,-178.593,6.212,148.705
C01156=1185.536,125.384,-52.846,-178.596,6.211,148.706
C01157=1185.541,125.134,-52.827,-178.599,6.209,148.706
C01158=1185.547,124.886,-52.807,-178.601,6.208,148.707
C01159=1185.551,124.637,-52.787,-178.604,6.206,148.707
C01160=1185.556,124.387,-52.767,-178.607,6.205,148.708
C01161=1185.560,124.137,-52.748,-178.609,6.204,148.708
C01162=1185.565,123.889,-52.729,-178.612,6.202,148.709
C01163=1185.569,123.640,-52.709,-178.615,6.201,148.709
C01164=1185.574,123.390,-52.689,-178.617,6.200,148.709
C01165=1185.580,123.141,-52.670,-178.620,6.198,148.710
C01166=1185.584,122.892,-52.650,-178.623,6.197,148.710
C01167=1185.589,122.642,-52.630,-178.625,6.196,148.711
C01168=1185.594,122.394,-52.610,-178.628,6.194,148.711
C01169=1185.599,122.145,-52.591,-178.631,6.192,148.712
C01170=1185.603,121.895,-52.572,-178.633,6.192,148.712
C01171=1185.608,121.646,-52.552,-178.636,6.190,148.713
C01172=1185.613,121.397,-52.533,-178.639,6.188,148.713
C01173=1185.618,121.147,-52.513,-178.641,6.187,148.714
C01174=1185.623,120.898,-52.494,-178.643,6.186,148.714
C01175=1185.628,120.649,-52.474,-178.646,6.185,148.715
C01176=1185.632,120.401,-52.455,-178.649,6.183,148.715
C01177=1185.637,120.151,-52.435,-178.651,6.182,148.716
C01178=1185.642,119.902,-52.415,-178.654,6.181,148.716
C01179=1185.647,119.653,-52.396,-178.657,6.179,148.717
C01180=1185.652,119.403,-52.376,-178.659,6.178,148.717
C01181=1185.656,119.154,-52.357,-178.662,6.177,148.718
C01182=1185.661,118.905,-52.338,-178.665,6.175,148.718
C01183=1185.666,118.656,-52.318,-178.667,6.174,148.718
C01184=1185.671,118.407,-52.299,-178.670,6.173,148.719
C01185=1185.675,118.158,-52.280,-178.673,6.171,148.719
C01186=1185.680,117.908,-52.260,-178.675,6.169,148.720
C01187=1185.685,117.659,-52.241,-178.678,6.169,148.720
C01188=1185.690,117.410,-52.222,-178.681,6.167,148.721
C01189=1185.694,117.161,-52.203,-178.683,6.166,148.721
C01190=1185.699,116.911,-52.183,-178.686,6.165,148.722
C01191=1185.705,116.663,-52.164,-178.689,6.163,148.722
C01192=1185.709,116.413,-52.146,-178.691,6.162,148.723
C01193=1185.714,116.164,-52.126,-178.694,6.161,148.723
C01194=1185.719,115.914,-52.107,-178.696,6.160,148.724
C01195=1185.723,115.665,-52.088,-178.699,6.158,148.724
C01196=1185.728,115.416,-52.068,-178.702,6.157,148.725
C01197=1185.733,115.167,-52.049,-178.704,6.156,148.725
C01198=1185.738,114.918,-52.030,-178.707,6.154,148.726
C01199=1185.742,114.668,-52.010,-178.710,6.153,148.726
C01200=1185.748,114.419,-51.992,-178.712,6.152,148.727
C01201=1185.752,114.170,-51.973,-178.715,6.150,148.727
C01202=1185.757,113.921,-51.953,-178.718,6.149,148.728
C01203=1185.762,113.671,-51.934,-178.720,6.148,148.728
C01204=1185.767,113.423,-51.915,-178.723,6.146,148.729
C01205=1185.772,113.173,-51.895,-178.726,6.145,148.729
C01206=1185.776,112.924,-51.877,-178.728,6.144,148.730
C01207=1185.781,112.674,-51.858,-178.731,6.143,148.730
C01208=1185.787,112.425,-51.838,-178.734,6.141,148.731
C01209=1185.791,112.176,-51.819,-178.736,6.140,148.731
C01210=1185.796,111.927,-51.801,-178.739,6.139,148.732
C01211=1185.800,111.677,-51.782,-178.742,6.137,148.732
C01212=1185.806,111.429,-51.762,-178.744,6.136,148.732
C01213=1185.810,111.179,-51.744,-178.747,6.135,148.733
C01214=1185.815,110.930,-51.725,-178.749,6.134,148.733
C01215=1185.821,110.681,-51.705,-178.752,6.132,148.734
C01216=1185.825,110.432,-51.686,-178.755,6.131,148.735
C01217=1185.830,110.182,-51.668,-178.757,6.130,148.735
C01218=1185.834,109.933,-51.649,-178.760,6.129,148.736
C01219=1185.840,109.684,-51.629,-178.762,6.128,148.736
C01220=1185.844,109.434,-51.611,-178.765,6.126,148.736
C01221=1185.849,109.185,-51.592,-178.768,6.125,148.737
C01222=1185.854,108.936,-51.574,-178.770,6.124,148.737
C01223=1185.859,108.687,-51.554,-178.773,6.122,148.738
C01224=1185.863,108.438,-51.536,-178.776,6.121,148.738
C01225=1185.868,108.188,-51.517,-178.778,6.120,148.739
C01226=1185.873,107.939,-51.498,-178.781,6.119,148.740
C01227=1185.877,107.689,-51.480,-178.784,6.117,148.740
C01228=1185.883,107.441,-51.460,-178.786,6.116,148.740
C01229=1185.887,107.192,-51.442,-178.789,6.115,148.741
C01230=1185.893,106.923,-51.421,-178.792,6.113,148.741
C01231=1185.898,106.654,-51.401,-178.795,6.112,148.742
C01232=1185.903,106.387,-51.381,-178.797,6.111,148.742
C01233=1185.908,106.117,-51.361,-178.800,6.110,148.743
C01234=1185.913,105.869,-51.342,-178.803,6.108,148.743
C01235=1185.919,105.619,-51.323,-178.806,6.107,148.744
C01236=1185.923,105.370,-51.304,-178.808,6.106,148.745
C01237=1185.928,105.121,-51.286,-178.811,6.105,148.745
C01238=1185.933,104.872,-51.267,-178.814,6.103,148.746
C01239=1185.937,104.622,-51.249,-178.816,6.102,148.746
C01240=1185.942,104.373,-51.231,-178.819,6.101,148.747
C01241=1185.947,104.124,-51.211,-178.821,6.100,148.747
C01242=1185.952,103.874,-51.193,-178.824,6.099,148.748
C01243=1185.956,103.626,-51.174,-178.826,6.098,148.748
C01244=1185.962,103.376,-51.156,-178.829,6.096,148.748
C01245=1185.966,103.127,-51.137,-178.832,6.095,148.749
C01246=1185.971,102.878,-51.119,-178.835,6.094,148.750
C01247=1185.977,102.628,-51.100,-178.838,6.092,148.750
C01248=1185.981,102.379,-51.081,-178.840,6.091,148.751
C01249=1185.986,102.130,-51.063,-178.843,6.090,148.751
C01250=1185.991,101.880,-51.045,-178.845,6.089,148.752
C01251=1185.995,101.631,-51.026,-178.848,6.087,148.752
C01252=1186.000,101.382,-51.008,-178.851,6.087,148.753
C01253=1186.006,101.132,-50.989,-178.853,6.085,148.753
C01254=1186.010,100.884,-50.970,-178.856,6.085,148.754
C01255=1186.015,100.634,-50.952,-178.859,6.083,148.754
C01256=1186.020,100.385,-50.934,-178.861,6.082,148.755
C01257=1186.025,100.135,-50.915,-178.864,6.081,148.755
C01258=1186.029,99.886,-50.896,-178.866,6.080,148.756
C01259=1186.034,99.637,-50.878,-178.869,6.078,148.756
C01260=1186.039,99.388,-50.860,-178.871,6.077,148.757
C01261=1186.045,99.138,-50.842,-178.875,6.076,148.757
C01262=1186.049,98.889,-50.823,-178.877,6.075,148.758
C01263=1186.054,98.640,-50.805,-178.879,6.073,148.758
C01264=1186.059,98.391,-50.787,-178.882,6.073,148.759
C01265=1186.063,98.141,-50.769,-178.885,6.071,148.759
C01266=1186.068,97.891,-50.750,-178.887,6.070,148.760
C01267=1186.073,97.643,-50.731,-178.890,6.069,148.760
C01268=1186.078,97.393,-50.713,-178.893,6.068,148.761
C01269=1186.083,97.144,-50.695,-178.895,6.066,148.761
C01270=1186.088,96.895,-50.677,-178.898,6.066,148.762
C01271=1186.092,96.645,-50.659,-178.901,6.064,148.762
C01272=1186.098,96.396,-50.640,-178.903,6.063,148.763
C01273=1186.102,96.147,-50.622,-178.906,6.062,148.763
C01274=1186.107,95.898,-50.604,-178.908,6.061,148.764
C01275=1186.112,95.649,-50.586,-178.911,6.060,148.765
C01276=1186.117,95.399,-50.567,-178.913,6.059,148.765
C01277=1186.121,95.150,-50.549,-178.917,6.057,148.766
C01278=1186.126,94.901,-50.531,-178.919,6.056,148.766
C01279=1186.131,94.651,-50.513,-178.922,6.055,148.767
C01280=1186.136,94.402,-50.495,-178.924,6.054,148.767
C01281=1186.142,94.153,-50.477,-178.927,6.052,148.767
C01282=1186.146,93.903,-50.458,-178.929,6.052,148.768
C01283=1186.151,93.654,-50.440,-178.932,6.050,148.769
C01284=1186.156,93.405,-50.423,-178.935,6.050,148.769
C01285=1186.161,93.155,-50.405,-178.938,6.048,148.770
C01286=1186.166,92.906,-50.387,-178.940,6.047,148.770
C01287=1186.171,92.657,-50.369,-178.943,6.046,148.771
C01288=1186.175,92.407,-50.350,-178.946,6.045,148.771
C01289=1186.180,92.158,-50.332,-178.948,6.044,148.772
C01290=1186.185,91.909,-50.314,-178.951,6.043,148.772
C01291=1186.190,91.660,-50.296,-178.953,6.042,148.773
C01292=1186.195,91.410,-50.278,-178.956,6.040,148.773
C01293=1186.200,91.161,-50.260,-178.958,6.039,148.774
C01294=1186.204,90.912,-50.242,-178.961,6.038,148.774
C01295=1186.209,90.663,-50.224,-178.964,6.037,148.775
C01296=1186.214,90.414,-50.206,-178.966,6.035,148.775
C01297=1186.219,90.163,-50.189,-178.969,6.035,148.776
C01298=1186.224,89.914,-50.171,-178.972,6.033,148.776
C01299=1186.229,89.665,-50.153,-178.974,6.033,148.777
C01300=1186.234,89.416,-50.135,-178.976,6.032,148.778
C01301=1186.239,89.167,-50.117,-178.980,6.030,148.778
C01302=1186.243,88.917,-50.099,-178.982,6.029,148.779
C01303=1186.248,88.668,-50.081,-178.985,6.028,148.779
C01304=1186.254,88.418,-50.064,-178.987,6.027,148.780
C01305=1186.259,88.169,-50.046,-178.990,6.026,148.780
C01306=1186.263,87.920,-50.028,-178.992,6.025,148.781
C01307=1186.268,87.671,-50.010,-178.996,6.024,148.781
C01308=1186.273,87.422,-49.992,-178.998,6.023,148.782
C01309=1186.278,87.172,-49.975,-179.000,6.022,148.782
C01310=1186.283,86.923,-49.957,-179.003,6.020,148.783
C01311=1186.288,86.674,-49.939,-179.006,6.020,148.783
C01312=1186.292,86.425,-49.921,-179.008,6.018,148.784
C01313=1186.297,86.174,-49.903,-179.011,6.018,148.785
C01314=1186.302,85.925,-49.885,-179.014,6.016,148.785
C01315=1186.307,85.676,-49.867,-179.016,6.015,148.786
C01316=1186.311,85.426,-49.851,-179.019,6.014,148.786
C01317=1186.316,85.177,-49.833,-179.022,6.013,148.787
C01318=1186.321,84.928,-49.815,-179.024,6.012,148.787
C01319=1186.326,84.678,-49.798,-179.027,6.011,148.788
C01320=1186.331,84.429,-49.780,-179.029,6.010,148.788
C01321=1186.336,84.180,-49.762,-179.032,6.009,148.789
C01322=1186.341,83.930,-49.745,-179.035,6.008,148.789
C01323=1186.346,83.681,-49.727,-179.037,6.007,148.790
C01324=1186.351,83.432,-49.709,-179.040,6.005,148.790
C01325=1186.356,83.182,-49.692,-179.043,6.005,148.791
C01326=1186.361,82.933,-49.674,-179.045,6.004,148.791
C01327=1186.365,82.685,-49.657,-179.048,6.002,148.792
C01328=1186.371,82.435,-49.639,-179.050,6.002,148.793
C01329=1186.376,82.186,-49.621,-179.053,6.000,148.793
C01330=1186.381,81.936,-49.604,-179.055,5.999,148.794
C01331=1186.386,81.687,-49.586,-179.059,5.998,148.794
C01332=1186.390,81.437,-49.570,-179.061,5.997,148.795
C01333=1186.395,81.188,-49.552,-179.063,5.997,148.795
C01334=1186.401,80.919,-49.533,-179.066,5.995,148.796
C01335=1186.406,80.651,-49.513,-179.069,5.994,148.796
C01336=1186.411,80.383,-49.496,-179.072,5.993,148.797
C01337=1186.416,80.115,-49.476,-179.075,5.991,148.797
C01338=1186.421,79.865,-49.459,-179.077,5.991,148.798
C01339=1186.426,79.616,-49.441,-179.080,5.990,148.799
C01340=1186.431,79.367,-49.424,-179.083,5.988,148.799
C01341=1186.436,79.117,-49.407,-179.085,5.988,148.800
C01342=1186.441,78.868,-49.389,-179.088,5.986,148.800
C01343=1186.445,78.618,-49.373,-179.091,5.986,148.801
C01344=1186.450,78.369,-49.355,-179.093,5.985,148.801
C01345=1186.456,78.120,-49.338,-179.096,5.983,148.802
C01346=1186.460,77.871,-49.320,-179.098,5.982,148.802
C01347=1186.465,77.621,-49.303,-179.101,5.982,148.803
C01348=1186.470,77.371,-49.286,-179.103,5.980,148.804
C01349=1186.475,77.123,-49.268,-179.106,5.980,148.804
C01350=1186.480,76.873,-49.251,-179.109,5.978,148.805
C01351=1186.485,76.624,-49.233,-179.111,5.977,148.805
C01352=1186.489,76.374,-49.216,-179.114,5.976,148.806
C01353=1186.495,76.125,-49.200,-179.117,5.975,148.806
C01354=1186.499,75.876,-49.182,-179.119,5.974,148.807
C01355=1186.504,75.626,-49.165,-179.122,5.974,148.807
C01356=1186.510,75.377,-49.148,-179.125,5.972,148.808
C01357=1186.514,75.128,-49.130,-179.127,5.971,148.809
C01358=1186.519,74.878,-49.113,-179.130,5.971,148.809
C01359=1186.524,74.629,-49.097,-179.132,5.969,148.810
C01360=1186.529,74.379,-49.079,-179.135,5.969,148.810
C01361=1186.534,74.130,-49.061,-179.137,5.968,148.811
C01362=1186.539,73.881,-49.045,-179.140,5.966,148.811
C01363=1186.544,73.631,-49.027,-179.142,5.965,148.812
C01364=1186.548,73.382,-49.010,-179.146,5.964,148.812
C01365=1186.554,73.133,-48.993,-179.148,5.963,148.813
C01366=1186.558,72.883,-48.977,-179.150,5.963,148.814
C01367=1186.564,72.634,-48.959,-179.154,5.961,148.814
C01368=1186.568,72.384,-48.943,-179.156,5.960,148.815
C01369=1186.573,72.135,-48.925,-179.158,5.960,148.815
C01370=1186.578,71.886,-48.908,-179.161,5.958,148.816
C01371=1186.583,71.636,-48.891,-179.164,5.958,148.816
C01372=1186.588,71.387,-48.874,-179.166,5.957,148.817
C01373=1186.593,71.137,-48.857,-179.169,5.955,148.817
C01374=1186.598,70.888,-48.841,-179.171,5.954,148.818
C01375=1186.603,70.639,-48.823,-179.174,5.954,148.819
C01376=1186.608,70.390,-48.806,-179.177,5.953,148.819
C01377=1186.613,70.140,-48.789,-179.179,5.952,148.820
C01378=1186.618,69.891,-48.773,-179.182,5.951,148.820
C01379=1186.622,69.642,-48.756,-179.185,5.949,148.821
C01380=1186.628,69.392,-48.739,-179.187,5.949,148.821
C01381=1186.632,69.142,-48.722,-179.189,5.948,148.822
C01382=1186.638,68.893,-48.705,-179.193,5.947,148.822
C01383=1186.642,68.644,-48.688,-179.195,5.946,148.823
C01384=1186.647,68.395,-48.670,-179.197,5.945,148.824
C01385=1186.652,68.145,-48.654,-179.200,5.945,148.824
C01386=1186.657,67.896,-48.637,-179.203,5.943,148.825
C01387=1186.662,67.646,-48.620,-179.205,5.942,148.825
C01388=1186.667,67.397,-48.604,-179.207,5.942,148.826
C01389=1186.672,67.147,-48.586,-179.211,5.940,148.826
C01390=1186.677,66.898,-48.570,-179.213,5.939,148.827
C01391=1186.681,66.649,-48.553,-179.215,5.939,148.827
C01392=1186.686,66.399,-48.536,-179.219,5.937,148.828
C01393=1186.692,66.150,-48.520,-179.221,5.937,148.829
C01394=1186.696,65.901,-48.503,-179.223,5.936,148.829
C01395=1186.701,65.651,-48.486,-179.226,5.934,148.830
C01396=1186.706,65.402,-48.470,-179.229,5.934,148.830
C01397=1186.711,65.152,-48.454,-179.231,5.933,148.831
C01398=1186.716,64.902,-48.436,-179.234,5.932,148.831
C01399=1186.721,64.654,-48.420,-179.237,5.931,148.832
C01400=1186.726,64.404,-48.403,-179.239,5.930,148.832
C01401=1186.731,64.154,-48.386,-179.242,5.930,148.833
C01402=1186.736,63.906,-48.370,-179.244,5.928,148.834
C01403=1186.741,63.656,-48.353,-179.247,5.927,148.834
C01404=1186.745,63.407,-48.336,-179.250,5.927,148.835
C01405=1186.751,63.158,-48.320,-179.252,5.926,148.835
C01406=1186.755,62.908,-48.303,-179.255,5.925,148.836
C01407=1186.760,62.658,-48.287,-179.257,5.924,148.836
C01408=1186.765,62.409,-48.271,-179.260,5.923,148.837
C01409=1186.771,62.159,-48.253,-179.263,5.922,148.838
C01410=1186.776,61.911,-48.237,-179.265,5.921,148.838
C01411=1186.780,61.661,-48.220,-179.268,5.920,148.839
C01412=1186.785,61.412,-48.204,-179.270,5.920,148.839
C01413=1186.791,61.162,-48.188,-179.273,5.918,148.840
C01414=1186.795,60.912,-48.171,-179.276,5.918,148.841
C01415=1186.800,60.664,-48.155,-179.278,5.917,148.841
C01416=1186.805,60.414,-48.138,-179.281,5.915,148.842
C01417=1186.810,60.164,-48.122,-179.283,5.915,148.842
C01418=1186.815,59.915,-48.105,-179.286,5.914,148.843
C01419=1186.820,59.665,-48.088,-179.288,5.913,148.843
C01420=1186.825,59.417,-48.072,-179.291,5.912,148.844
C01421=1186.830,59.167,-48.056,-179.294,5.911,148.845
C01422=1186.834,58.917,-48.039,-179.296,5.910,148.845
C01423=1186.840,58.668,-48.023,-179.299,5.910,148.846
C01424=1186.845,58.418,-48.007,-179.302,5.908,148.846
C01425=1186.850,58.169,-47.990,-179.304,5.908,148.847
C01426=1186.854,57.920,-47.974,-179.307,5.907,148.847
C01427=1186.859,57.671,-47.957,-179.309,5.906,148.848
C01428=1186.864,57.421,-47.941,-179.312,5.905,148.849
C01429=1186.869,57.172,-47.925,-179.315,5.904,148.849
C01430=1186.875,56.922,-47.908,-179.317,5.903,148.850
C01431=1186.880,56.673,-47.892,-179.319,5.903,148.850
C01432=1186.884,56.423,-47.876,-179.322,5.901,148.851
C01433=1186.890,56.174,-47.860,-179.325,5.901,148.851
C01434=1186.894,55.924,-47.843,-179.327,5.900,148.852
C01435=1186.899,55.676,-47.827,-179.330,5.899,148.853
C01436=1186.904,55.425,-47.811,-179.333,5.898,148.853
C01437=1186.909,55.177,-47.795,-179.335,5.897,148.854
C01438=1186.914,54.908,-47.777,-179.338,5.897,148.854
C01439=1186.920,54.639,-47.760,-179.341,5.895,148.855
C01440=1186.926,54.371,-47.742,-179.343,5.895,148.856
C01441=1186.931,54.102,-47.725,-179.346,5.894,148.856
C01442=1186.936,53.853,-47.708,-179.349,5.892,148.857
C01443=1186.941,53.603,-47.692,-179.351,5.892,148.857
C01444=1186.946,53.354,-47.676,-179.354,5.891,148.858
C01445=1186.950,53.104,-47.660,-179.356,5.891,148.859
C01446=1186.955,52.855,-47.644,-179.359,5.889,148.859
C01447=1186.960,52.605,-47.628,-179.362,5.888,148.860
C01448=1186.965,52.356,-47.612,-179.364,5.888,148.860
C01449=1186.971,52.107,-47.596,-179.367,5.887,148.861
C01450=1186.976,51.857,-47.580,-179.370,5.886,148.861
C01451=1186.981,51.608,-47.564,-179.372,5.885,148.862
C01452=1186.985,51.358,-47.548,-179.375,5.885,148.863
C01453=1186.990,51.109,-47.531,-179.377,5.884,148.863
C01454=1186.995,50.859,-47.515,-179.380,5.883,148.864
C01455=1187.000,50.610,-47.499,-179.383,5.882,148.864
C01456=1187.005,50.360,-47.483,-179.385,5.881,148.865
C01457=1187.011,50.111,-47.468,-179.388,5.880,148.866
C01458=1187.016,49.862,-47.451,-179.390,5.880,148.866
C01459=1187.020,49.612,-47.436,-179.392,5.879,148.867
C01460=1187.025,49.363,-47.420,-179.396,5.878,148.867
C01461=1187.030,49.113,-47.404,-179.398,5.877,148.868
C01462=1187.035,48.864,-47.388,-179.400,5.876,148.868
C01463=1187.039,48.614,-47.371,-179.403,5.876,148.869
C01464=1187.045,48.365,-47.356,-179.405,5.875,148.870
C01465=1187.050,48.116,-47.340,-179.408,5.874,148.870
C01466=1187.055,47.866,-47.324,-179.411,5.873,148.871
C01467=1187.060,47.617,-47.308,-179.413,5.872,148.871
C01468=1187.065,47.367,-47.292,-179.416,5.872,148.872
C01469=1187.069,47.117,-47.277,-179.418,5.871,148.873
C01470=1187.075,46.869,-47.261,-179.421,5.869,148.873
C01471=1187.079,46.619,-47.245,-179.424,5.869,148.874
C01472=1187.085,46.369,-47.229,-179.426,5.868,148.874
C01473=1187.090,46.120,-47.213,-179.429,5.867,148.875
C01474=1187.095,45.870,-47.197,-179.431,5.867,148.876
C01475=1187.100,45.621,-47.181,-179.434,5.865,148.876
C01476=1187.105,45.372,-47.166,-179.437,5.865,148.877
C01477=1187.109,45.122,-47.150,-179.439,5.864,148.877
C01478=1187.114,44.873,-47.134,-179.441,5.863,148.878
C01479=1187.120,44.623,-47.119,-179.444,5.863,148.879
C01480=1187.125,44.373,-47.103,-179.447,5.862,148.879
C01481=1187.129,44.124,-47.088,-179.449,5.861,148.880
C01482=1187.135,43.875,-47.072,-179.452,5.860,148.880
C01483=1187.139,43.625,-47.055,-179.455,5.860,148.881
C01484=1187.145,43.376,-47.040,-179.457,5.859,148.881
C01485=1187.150,43.127,-47.024,-179.460,5.858,148.882
C01486=1187.154,42.877,-47.009,-179.463,5.857,148.883
C01487=1187.159,42.627,-46.993,-179.465,5.856,148.883
C01488=1187.165,42.378,-46.978,-179.468,5.856,148.884
C01489=1187.170,42.129,-46.962,-179.470,5.855,148.884
C01490=1187.174,41.879,-46.947,-179.472,5.854,148.885
C01491=1187.179,41.630,-46.930,-179.475,5.854,148.886
C01492=1187.185,41.381,-46.915,-179.478,5.852,148.886
C01493=1187.189,41.131,-46.899,-179.480,5.851,148.887
C01494=1187.194,40.881,-46.884,-179.483,5.851,148.887
C01495=1187.199,40.632,-46.868,-179.485,5.850,148.888
C01496=1187.205,40.383,-46.853,-179.488,5.849,148.889
C01497=1187.209,40.133,-46.837,-179.490,5.849,148.889
C01498=1187.214,39.883,-46.822,-179.493,5.848,148.890
C01499=1187.220,39.634,-46.806,-179.496,5.847,148.890
C01500=1187.224,39.385,-46.791,-179.498,5.846,148.891
C01501=1187.229,39.135,-46.775,-179.501,5.845,148.891
C01502=1187.235,38.885,-46.760,-179.503,5.845,148.892
C01503=1187.239,38.636,-46.745,-179.506,5.844,148.893
C01504=1187.245,38.387,-46.729,-179.508,5.843,148.893
C01505=1187.249,38.137,-46.713,-179.511,5.843,148.894
C01506=1187.254,37.888,-46.698,-179.514,5.842,148.895
C01507=1187.259,37.638,-46.682,-179.516,5.841,148.895
C01508=1187.265,37.389,-46.667,-179.519,5.840,148.896
C01509=1187.269,37.140,-46.652,-179.521,5.840,148.896
C01510=1187.274,36.890,-46.636,-179.524,5.839,148.897
C01511=1187.280,36.640,-46.620,-179.526,5.838,148.898
C01512=1187.285,36.391,-46.606,-179.529,5.838,148.898
C01513=1187.290,36.141,-46.590,-179.532,5.836,148.899
C01514=1187.295,35.892,-46.575,-179.534,5.836,148.899
C01515=1187.299,35.642,-46.560,-179.537,5.835,148.900
C01516=1187.305,35.393,-46.544,-179.539,5.835,148.901
C01517=1187.309,35.144,-46.529,-179.542,5.834,148.901
C01518=1187.315,34.894,-46.513,-179.544,5.833,148.902
C01519=1187.319,34.645,-46.498,-179.547,5.833,148.902
C01520=1187.325,34.395,-46.483,-179.549,5.832,148.903
C01521=1187.329,34.145,-46.468,-179.552,5.831,148.904
C01522=1187.335,33.896,-46.453,-179.555,5.830,148.904
C01523=1187.340,33.646,-46.437,-179.557,5.829,148.905
C01524=1187.345,33.397,-46.422,-179.560,5.829,148.905
C01525=1187.350,33.148,-46.406,-179.562,5.828,148.906
C01526=1187.355,32.898,-46.392,-179.565,5.827,148.907
C01527=1187.360,32.648,-46.376,-179.567,5.827,148.907
C01528=1187.364,32.399,-46.361,-179.570,5.826,148.908
C01529=1187.370,32.150,-46.346,-179.572,5.825,148.908
C01530=1187.375,31.900,-46.331,-179.575,5.824,148.909
C01531=1187.380,31.651,-46.316,-179.578,5.824,148.910
C01532=1187.385,31.401,-46.301,-179.580,5.823,148.910
C01533=1187.390,31.152,-46.285,-179.583,5.822,148.911
C01534=1187.395,30.902,-46.271,-179.585,5.822,148.911
C01535=1187.400,30.652,-46.255,-179.587,5.821,148.912
C01536=1187.405,30.403,-46.240,-179.590,5.820,148.913
C01537=1187.409,30.153,-46.226,-179.593,5.820,148.913
C01538=1187.415,29.904,-46.210,-179.595,5.819,148.914
C01539=1187.420,29.655,-46.195,-179.598,5.818,148.914
C01540=1187.425,29.405,-46.180,-179.601,5.817,148.915
C01541=1187.430,29.156,-46.165,-179.603,5.817,148.916
C01542=1187.436,28.887,-46.149,-179.606,5.816,148.916
C01543=1187.441,28.619,-46.132,-179.608,5.815,148.917
C01544=1187.446,28.349,-46.116,-179.611,5.815,148.918
C01545=1187.452,28.081,-46.100,-179.614,5.814,148.918
C01546=1187.457,27.831,-46.085,-179.617,5.813,148.919
C01547=1187.462,27.582,-46.071,-179.619,5.813,148.920
C01548=1187.467,27.332,-46.056,-179.622,5.812,148.920
C01549=1187.472,27.082,-46.041,-179.624,5.811,148.921
C01550=1187.477,26.833,-46.026,-179.627,5.811,148.921
C01551=1187.482,26.584,-46.011,-179.629,5.810,148.922
C01552=1187.487,26.334,-45.996,-179.632,5.809,148.923
C01553=1187.492,26.085,-45.981,-179.634,5.809,148.923
C01554=1187.497,25.834,-45.966,-179.637,5.808,148.924
C01555=1187.502,25.585,-45.951,-179.639,5.807,148.924
C01556=1187.507,25.336,-45.936,-179.642,5.806,148.925
C01557=1187.512,25.086,-45.921,-179.645,5.806,148.926
C01558=1187.517,24.836,-45.906,-179.647,5.805,148.926
C01559=1187.522,24.587,-45.892,-179.650,5.804,148.927
C01560=1187.527,24.337,-45.877,-179.652,5.804,148.928
C01561=1187.532,24.088,-45.862,-179.655,5.803,148.928
C01562=1187.537,23.839,-45.847,-179.657,5.802,148.929
C01563=1187.541,23.589,-45.832,-179.660,5.802,148.929
C01564=1187.547,23.339,-45.817,-179.663,5.801,148.930
C01565=1187.552,23.090,-45.803,-179.665,5.800,148.930
C01566=1187.557,22.841,-45.788,-179.667,5.800,148.931
C01567=1187.562,22.591,-45.773,-179.670,5.800,148.932
C01568=1187.567,22.342,-45.758,-179.672,5.799,148.932
C01569=1187.572,22.092,-45.744,-179.675,5.798,148.933
C01570=1187.577,21.843,-45.729,-179.677,5.798,148.934
C01571=1187.583,21.593,-45.715,-179.680,5.797,148.934
C01572=1187.588,21.344,-45.700,-179.683,5.795,148.935
C01573=1187.593,21.095,-45.685,-179.686,5.795,148.935
C01574=1187.598,20.845,-45.671,-179.688,5.794,148.936
C01575=1187.603,20.595,-45.655,-179.690,5.794,148.937
C01576=1187.608,20.346,-45.641,-179.693,5.793,148.937
C01577=1187.613,20.096,-45.627,-179.696,5.793,148.938
C01578=1187.618,19.847,-45.612,-179.698,5.792,148.938
C01579=1187.622,19.597,-45.598,-179.700,5.791,148.939
C01580=1187.628,19.347,-45.583,-179.703,5.791,148.940
C01581=1187.633,19.098,-45.568,-179.706,5.790,148.940
C01582=1187.638,18.848,-45.553,-179.708,5.789,148.941
C01583=1187.643,18.599,-45.539,-179.711,5.789,148.942
C01584=1187.647,18.350,-45.524,-179.713,5.788,148.942
C01585=1187.652,18.100,-45.510,-179.715,5.788,148.943
C01586=1187.659,17.851,-45.495,-179.718,5.787,148.943
C01587=1187.664,17.601,-45.481,-179.721,5.787,148.944
C01588=1187.668,17.352,-45.466,-179.723,5.786,148.945
C01589=1187.673,17.102,-45.452,-179.725,5.785,148.945
C01590=1187.678,16.852,-45.438,-179.728,5.785,148.946
C01591=1187.683,16.603,-45.423,-179.731,5.784,148.947
C01592=1187.688,16.354,-45.408,-179.733,5.783,148.947
C01593=1187.693,16.104,-45.393,-179.736,5.783,148.948
C01594=1187.698,15.854,-45.379,-179.738,5.782,148.948
C01595=1187.704,15.605,-45.365,-179.741,5.782,148.949
C01596=1187.709,15.355,-45.351,-179.743,5.781,148.950
C01597=1187.714,15.106,-45.336,-179.746,5.781,148.950
C01598=1187.719,14.856,-45.322,-179.748,5.780,148.951
C01599=1187.723,14.607,-45.307,-179.751,5.780,148.952
C01600=1187.728,14.357,-45.293,-179.753,5.779,148.952
C01601=1187.733,14.107,-45.279,-179.756,5.778,148.953
C01602=1187.739,13.858,-45.265,-179.758,5.778,148.953
C01603=1187.744,13.609,-45.250,-179.761,5.777,148.954
C01604=1187.749,13.359,-45.235,-179.763,5.776,148.955
C01605=1187.754,13.109,-45.221,-179.766,5.776,148.955
C01606=1187.759,12.860,-45.207,-179.769,5.775,148.956
C01607=1187.764,12.610,-45.192,-179.771,5.774,148.956
C01608=1187.770,12.361,-45.178,-179.774,5.773,148.957
C01609=1187.775,12.111,-45.164,-179.777,5.773,148.958
C01610=1187.780,11.862,-45.150,-179.779,5.772,148.958
C01611=1187.785,11.612,-45.136,-179.781,5.771,148.959
C01612=1187.790,11.362,-45.121,-179.784,5.771,148.960
C01613=1187.795,11.113,-45.107,-179.787,5.770,148.960
C01614=1187.800,10.863,-45.093,-179.789,5.770,148.961
C01615=1187.805,10.614,-45.079,-179.792,5.769,148.961
C01616=1187.810,10.364,-45.065,-179.794,5.769,148.962
C01617=1187.815,10.114,-45.050,-179.796,5.769,148.963
C01618=1187.820,9.865,-45.036,-179.798,5.768,148.963
C01619=1187.825,9.616,-45.022,-179.801,5.768,148.964
C01620=1187.830,9.366,-45.008,-179.804,5.767,148.965
C01621=1187.835,9.116,-44.994,-179.806,5.767,148.965
C01622=1187.841,8.867,-44.980,-179.809,5.766,148.966
C01623=1187.845,8.618,-44.966,-179.811,5.765,148.966
C01624=1187.850,8.368,-44.952,-179.814,5.765,148.967
C01625=1187.855,8.118,-44.937,-179.816,5.764,148.968
C01626=1187.860,7.869,-44.923,-179.819,5.763,148.968
C01627=1187.865,7.620,-44.909,-179.821,5.763,148.969
C01628=1187.870,7.370,-44.895,-179.824,5.762,148.970
C01629=1187.875,7.120,-44.881,-179.826,5.762,148.970
C01630=1187.881,6.871,-44.867,-179.829,5.761,148.971
C01631=1187.886,6.621,-44.852,-179.831,5.761,148.971
C01632=1187.891,6.372,-44.838,-179.834,5.760,148.972
C01633=1187.896,6.122,-44.824,-179.836,5.759,148.973
C01634=1187.901,5.873,-44.811,-179.839,5.759,148.973
C01635=1187.906,5.623,-44.797,-179.842,5.758,148.974
C01636=1187.911,5.373,-44.783,-179.844,5.758,148.975
C01637=1187.916,5.124,-44.768,-179.846,5.757,148.975
C01638=1187.921,4.875,-44.755,-179.849,5.757,148.976
C01639=1187.926,4.625,-44.740,-179.852,5.756,148.976
C01640=1187.931,4.375,-44.726,-179.854,5.756,148.977
C01641=1187.936,4.126,-44.713,-179.856,5.755,148.978
C01642=1187.941,3.876,-44.699,-179.859,5.754,148.978
C01643=1187.946,3.626,-44.685,-179.862,5.754,148.979
C01644=1187.952,3.377,-44.671,-179.864,5.753,148.979
C01645=1187.957,3.128,-44.657,-179.867,5.752,148.980
C01646=1187.962,2.858,-44.642,-179.869,5.752,148.981
C01647=1187.968,2.589,-44.627,-179.872,5.751,148.982
C01648=1187.974,2.320,-44.612,-179.875,5.751,148.982
C01649=1187.978,2.051,-44.598,-179.877,5.750,148.983
C01650=1187.983,1.801,-44.583,-179.880,5.750,148.984
C01651=1187.989,1.551,-44.570,-179.883,5.750,148.984
C01652=1187.994,1.302,-44.556,-179.885,5.749,148.985
C01653=1187.999,1.052,-44.542,-179.887,5.748,148.985
C01654=1188.004,0.804,-44.528,-179.890,5.748,148.986
C01655=1188.009,0.553,-44.515,-179.892,5.747,148.987
C01656=1188.014,0.304,-44.500,-179.895,5.746,148.987
C01657=1188.020,0.055,-44.487,-179.897,5.746,148.988
C01658=1188.024,-0.196,-44.474,-179.900,5.745,148.989
C01659=1188.029,-0.445,-44.459,-179.902,5.745,148.989
C01660=1188.035,-0.694,-44.445,-179.905,5.744,148.990
C01661=1188.040,-0.945,-44.432,-179.908,5.744,148.990
C01662=1188.045,-1.193,-44.418,-179.910,5.744,148.991
C01663=1188.050,-1.443,-44.404,-179.912,5.743,148.992
C01664=1188.055,-1.693,-44.391,-179.915,5.743,148.992
C01665=1188.060,-1.942,-44.377,-179.917,5.742,148.993
C01666=1188.065,-2.192,-44.364,-179.920,5.742,148.994
C01667=1188.071,-2.441,-44.350,-179.922,5.741,148.994
C01668=1188.075,-2.691,-44.336,-179.925,5.740,148.995
C01669=1188.080,-2.941,-44.323,-179.927,5.740,148.996
C01670=1188.086,-3.190,-44.309,-179.930,5.739,148.996
C01671=1188.090,-3.440,-44.296,-179.932,5.739,148.997
C01672=1188.096,-3.689,-44.282,-179.935,5.738,148.997
C01673=1188.101,-3.939,-44.268,-179.937,5.738,148.998
C01674=1188.106,-4.188,-44.255,-179.940,5.737,148.999
C01675=1188.111,-4.438,-44.241,-179.942,5.736,148.999
C01676=1188.116,-4.688,-44.227,-179.944,5.737,149.000
C01677=1188.121,-4.937,-44.214,-179.947,5.736,149.001
C01678=1188.126,-5.187,-44.200,-179.950,5.736,149.001
C01679=1188.132,-5.436,-44.186,-179.952,5.735,149.002
C01680=1188.136,-5.686,-44.173,-179.954,5.734,149.002
C01681=1188.142,-5.935,-44.159,-179.957,5.734,149.003
C01682=1188.146,-6.185,-44.146,-179.960,5.733,149.004
C01683=1188.152,-6.434,-44.133,-179.962,5.733,149.004
C01684=1188.157,-6.685,-44.119,-179.965,5.732,149.005
C01685=1188.162,-6.934,-44.106,-179.967,5.732,149.006
C01686=1188.167,-7.184,-44.092,-179.970,5.731,149.006
C01687=1188.172,-7.434,-44.079,-179.971,5.731,149.007
C01688=1188.177,-7.683,-44.065,-179.974,5.731,149.008
C01689=1188.182,-7.933,-44.052,-179.977,5.730,149.008
C01690=1188.187,-8.182,-44.038,-179.979,5.730,149.009
C01691=1188.192,-8.432,-44.025,-179.982,5.729,149.009
C01692=1188.198,-8.681,-44.012,-179.984,5.728,149.010
C01693=1188.203,-8.931,-43.998,-179.987,5.728,149.011
C01694=1188.208,-9.180,-43.985,-179.990,5.727,149.011
C01695=1188.213,-9.430,-43.971,-179.992,5.727,149.012
C01696=1188.218,-9.679,-43.958,-179.994,5.726,149.013
C01697=1188.223,-9.930,-43.945,-179.996,5.726,149.013
C01698=1188.228,-10.178,-43.932,-179.999,5.726,149.014
C01699=1188.234,-10.428,-43.918,179.999,5.725,149.014
C01700=1188.238,-10.678,-43.905,179.996,5.725,149.015
C01701=1188.244,-10.927,-43.892,179.993,5.724,149.016
C01702=1188.248,-11.177,-43.879,179.991,5.724,149.017
C01703=1188.254,-11.427,-43.865,179.989,5.723,149.017
C01704=1188.259,-11.676,-43.852,179.986,5.722,149.018
C01705=1188.264,-11.926,-43.838,179.983,5.722,149.018
C01706=1188.269,-12.176,-43.825,179.981,5.722,149.019
C01707=1188.274,-12.425,-43.813,179.979,5.721,149.020
C01708=1188.279,-12.675,-43.799,179.976,5.721,149.020
C01709=1188.284,-12.924,-43.786,179.974,5.720,149.021
C01710=1188.290,-13.174,-43.773,179.971,5.720,149.022
C01711=1188.294,-13.423,-43.759,179.969,5.719,149.022
C01712=1188.300,-13.673,-43.746,179.966,5.719,149.023
C01713=1188.305,-13.923,-43.733,179.964,5.718,149.023
C01714=1188.310,-14.172,-43.720,179.961,5.719,149.024
C01715=1188.315,-14.422,-43.707,179.959,5.718,149.025
C01716=1188.320,-14.671,-43.694,179.957,5.717,149.025
C01717=1188.326,-14.921,-43.680,179.954,5.717,149.026
C01718=1188.330,-15.171,-43.667,179.951,5.716,149.027
C01719=1188.336,-15.420,-43.654,179.949,5.715,149.027
C01720=1188.341,-15.670,-43.641,179.946,5.715,149.028
C01721=1188.345,-15.919,-43.628,179.944,5.715,149.029
C01722=1188.351,-16.169,-43.615,179.942,5.715,149.029
C01723=1188.356,-16.419,-43.602,179.940,5.714,149.030
C01724=1188.361,-16.668,-43.589,179.937,5.714,149.030
C01725=1188.367,-16.918,-43.576,179.934,5.713,149.031
C01726=1188.371,-17.168,-43.563,179.932,5.713,149.032
C01727=1188.376,-17.417,-43.550,179.929,5.712,149.032
C01728=1188.381,-17.667,-43.536,179.927,5.711,149.033
C01729=1188.386,-17.916,-43.523,179.925,5.712,149.034
C01730=1188.392,-18.166,-43.510,179.922,5.711,149.034
C01731=1188.397,-18.416,-43.497,179.919,5.711,149.035
C01732=1188.402,-18.665,-43.485,179.917,5.710,149.036
C01733=1188.407,-18.914,-43.472,179.915,5.709,149.036
C01734=1188.412,-19.165,-43.459,179.912,5.709,149.037
C01735=1188.418,-19.414,-43.446,179.909,5.709,149.038
C01736=1188.423,-19.663,-43.433,179.908,5.709,149.038
C01737=1188.428,-19.914,-43.420,179.905,5.708,149.039
C01738=1188.433,-20.163,-43.407,179.902,5.708,149.039
C01739=1188.438,-20.412,-43.395,179.900,5.707,149.040
C01740=1188.443,-20.663,-43.381,179.897,5.706,149.041
C01741=1188.449,-20.912,-43.368,179.895,5.706,149.041
C01742=1188.454,-21.161,-43.356,179.893,5.706,149.042
C01743=1188.458,-21.411,-43.343,179.890,5.706,149.043
C01744=1188.464,-21.661,-43.330,179.888,5.705,149.043
C01745=1188.469,-21.910,-43.317,179.885,5.704,149.044
C01746=1188.474,-22.160,-43.304,179.883,5.704,149.045
C01747=1188.479,-22.410,-43.291,179.880,5.703,149.045
C01748=1188.485,-22.659,-43.278,179.878,5.703,149.046
C01749=1188.490,-22.909,-43.266,179.876,5.703,149.046
C01750=1188.495,-23.178,-43.252,179.873,5.703,149.047
C01751=1188.501,-23.448,-43.238,179.870,5.702,149.048
C01752=1188.506,-23.717,-43.224,179.868,5.702,149.049
C01753=1188.512,-23.987,-43.210,179.865,5.701,149.049
C01754=1188.517,-24.237,-43.198,179.862,5.701,149.050
C01755=1188.522,-24.486,-43.185,179.860,5.700,149.051
C01756=1188.527,-24.736,-43.172,179.858,5.699,149.051
C01757=1188.532,-24.985,-43.159,179.855,5.699,149.052
C01758=1188.538,-25.236,-43.147,179.853,5.699,149.052
C01759=1188.543,-25.485,-43.134,179.850,5.699,149.053
C01760=1188.548,-25.735,-43.121,179.848,5.698,149.054
C01761=1188.553,-25.984,-43.109,179.845,5.698,149.054
C01762=1188.558,-26.234,-43.096,179.843,5.697,149.055
C01763=1188.563,-26.483,-43.084,179.841,5.697,149.056
C01764=1188.567,-26.733,-43.071,179.838,5.697,149.056
C01765=1188.574,-26.983,-43.058,179.836,5.696,149.057
C01766=1188.579,-27.232,-43.045,179.833,5.696,149.058
C01767=1188.584,-27.482,-43.033,179.830,5.695,149.058
C01768=1188.588,-27.732,-43.020,179.828,5.694,149.059
C01769=1188.594,-27.981,-43.007,179.826,5.695,149.059
C01770=1188.599,-28.231,-42.995,179.824,5.694,149.060
C01771=1188.604,-28.480,-42.983,179.821,5.694,149.061
C01772=1188.609,-28.730,-42.970,179.819,5.693,149.061
C01773=1188.614,-28.980,-42.957,179.816,5.693,149.062
C01774=1188.620,-29.230,-42.945,179.814,5.693,149.063
C01775=1188.625,-29.479,-42.932,179.811,5.692,149.063
C01776=1188.630,-29.729,-42.920,179.809,5.692,149.064
C01777=1188.635,-29.978,-42.907,179.806,5.691,149.065
C01778=1188.640,-30.229,-42.895,179.804,5.691,149.065
C01779=1188.645,-30.478,-42.882,179.802,5.691,149.066
C01780=1188.650,-30.727,-42.870,179.800,5.690,149.066
C01781=1188.655,-30.976,-42.857,179.797,5.690,149.067
C01782=1188.661,-31.226,-42.845,179.794,5.689,149.068
C01783=1188.666,-31.476,-42.832,179.792,5.689,149.069
C01784=1188.671,-31.726,-42.819,179.790,5.689,149.069
C01785=1188.676,-31.976,-42.808,179.787,5.688,149.070
C01786=1188.681,-32.225,-42.795,179.785,5.688,149.070
C01787=1188.686,-32.474,-42.782,179.782,5.687,149.071
C01788=1188.692,-32.724,-42.770,179.780,5.687,149.072
C01789=1188.697,-32.974,-42.758,179.778,5.687,149.072
C01790=1188.702,-33.224,-42.746,179.775,5.687,149.073
C01791=1188.707,-33.474,-42.733,179.772,5.686,149.074
C01792=1188.712,-33.723,-42.720,179.770,5.685,149.074
C01793=1188.717,-33.973,-42.709,179.768,5.686,149.075
C01794=1188.722,-34.222,-42.696,179.765,5.685,149.076
C01795=1188.728,-34.471,-42.683,179.763,5.685,149.076
C01796=1188.733,-34.721,-42.671,179.760,5.684,149.077
C01797=1188.738,-34.971,-42.659,179.758,5.683,149.077
C01798=1188.744,-35.221,-42.647,179.756,5.684,149.078
C01799=1188.749,-35.470,-42.634,179.753,5.683,149.079
C01800=1188.753,-35.721,-42.622,179.751,5.683,149.079
C01801=1188.759,-35.970,-42.610,179.748,5.682,149.080
C01802=1188.764,-36.220,-42.598,179.746,5.682,149.081
C01803=1188.769,-36.469,-42.585,179.744,5.682,149.081
C01804=1188.774,-36.718,-42.572,179.741,5.682,149.082
C01805=1188.780,-36.968,-42.561,179.739,5.681,149.083
C01806=1188.784,-37.217,-42.549,179.736,5.680,149.083
C01807=1188.790,-37.467,-42.537,179.734,5.681,149.084
C01808=1188.795,-37.717,-42.524,179.731,5.680,149.085
C01809=1188.800,-37.967,-42.512,179.729,5.679,149.085
C01810=1188.805,-38.216,-42.500,179.727,5.679,149.086
C01811=1188.811,-38.466,-42.488,179.724,5.679,149.086
C01812=1188.816,-38.716,-42.476,179.722,5.679,149.087
C01813=1188.821,-38.965,-42.463,179.720,5.678,149.088
C01814=1188.827,-39.215,-42.451,179.717,5.678,149.088
C01815=1188.830,-39.465,-42.439,179.715,5.678,149.089
C01816=1188.836,-39.715,-42.427,179.712,5.677,149.090
C01817=1188.841,-39.964,-42.414,179.710,5.677,149.090
C01818=1188.846,-40.214,-42.403,179.707,5.676,149.091
C01819=1188.852,-40.464,-42.391,179.705,5.676,149.092
C01820=1188.857,-40.713,-42.378,179.703,5.676,149.092
